KUKA KRL program: EPS_2_25694_GD03_A_20260114065902.src

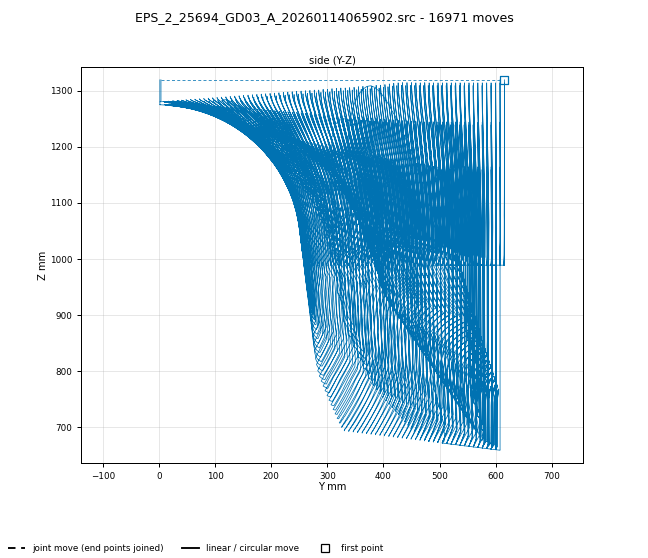
[picture p0: tool path of EPS_2_25694_GD03_A_20260114065902.src, 16971 of 16973 moves have a stored position in this frame; points joined in program order, loops and branches not executed]
&ACCESS RVP
&REL 4
&COMMENT QRS 19112012
&PARAM EDITMASK = *
DEF PART()
EXT BAS (BAS_COMMAND :IN,REAL :IN )
INT I
BAS (#INITMOV,0 )

;KUKA QRS Post kuka4.cps  Date:22-06-2017 !

File_ID=2970

QRS_PRE_INIT()

;Init var - Until changes are made in qrs_pre_init
Outlet_Square_prg=0
Inlet_1_Square_prg=0
Inlet_2_Square_prg=0
Inlet_3_Square_prg=0
Inlet_4_Square_prg=0
Inlet_5_Square_prg=0

Outlet_1={X 0.000, Y 425.000, Z 1043.000, B 0.000, E1 0.000 }
Inlet_1={X 0.000, Y 466.000, Z 1011.000, B 0.000, E1 180.000 }
Inlet_2={X 0.000, Y 490.880, Z 930.000, B 0.000, E1 271.000 }
Outlet_1_type=533
Inlet_1_type=457
Inlet_2_type=299
;QRS#1=Sidecore dimensions
;QRS#2=525-21" Concrete
;QRS#3=450-18" Concrete
;QRS#4=300-12" PVC SDR 35
;QRS#5=
;QRS#6=
;QRS#7=
;QRS#8=
;QRS#9=S306-32
;QRS#10=28A PSX-2
;QRS#11=16M PSX
;QRS#12=
;QRS#13=
;QRS#14=
;QRS#15=
;QRS#16=1220x127x1676 5,5'
;QRS#17=EPS Height
;QRS#18=1309,5
;QRS#19=*
;QRS#20= UPDATED VERSION 22-06-2017
;QRS#21=*
Outlet_Square=0250
Inlet_1_Square=0250
Inlet_2_Square=0150
Inlet_3_Square=0
Inlet_4_Square=0
Inlet_5_Square=0
Mill_Square=1
Outlet_Square_Prg=263
Inlet_1_Square_prg=274
Inlet_2_Square_prg=206

QRS_INIT()

$ADVANCE=5

; T1
PTP {E1 172.532,E2 172.532}
PTP {X 0,Y 615.614,A -85,B 0,C 180,E1 172.532,E2 172.532,E3 0,E4 0,E5 0,E6 0}
QRS_SPEED_INIT()
LIN {X 0,Y 615.614,Z 1319.5,A -85,B 0,C 180,E1 172.532,E2 172.532,E3 0,E4 0,E5 0,E6 0} C_VEL
LIN {X 0,Y 615.614,Z 991.03,A -85,B 0,C 180,E1 172.532,E2 172.532} C_VEL
LIN {X 0,Y 615.559,Z 989.03,A -85,B 0,C 180,E1 172.718,E2 172.718} C_VEL
LIN {X 0,Y 615.859,Z 989.03,A -85,B 0,C 180,E1 176.52,E2 176.52} C_VEL
LIN {X 0,Y 615.859,Z 989.03,A -85,B 0,C 180,E1 181.159,E2 181.159} C_VEL
LIN {X 0,Y 615.851,Z 989.03,A -85,B 0,C 180,E1 185.807,E2 185.807} C_VEL
LIN {X 0,Y 615.828,Z 989.03,A -85,B 0,C 180,E1 190.493,E2 190.493} C_VEL
LIN {X 0,Y 615.82,Z 989.03,A -85,B 0,C 180,E1 195.252,E2 195.252} C_VEL
LIN {X 0,Y 615.788,Z 989.03,A -85,B 0,C 180,E1 200.122,E2 200.122} C_VEL
LIN {X 0,Y 615.781,Z 989.03,A -85,B 0,C 180,E1 205.149,E2 205.149} C_VEL
LIN {X 0,Y 615.249,Z 989.03,A -85,B 0,C 180,E1 207.765,E2 207.765} C_VEL
LIN {X 0,Y 615.753,Z 989.03,A -85,B 0,C 180,E1 210.394,E2 210.394} C_VEL
LIN {X 0,Y 615.151,Z 989.03,A -85,B 0,C 180,E1 213.846,E2 213.846} C_VEL
LIN {X 0,Y 615.688,Z 989.03,A -85,B 0,C 180,E1 215.941,E2 215.941} C_VEL
LIN {X 0,Y 615.425,Z 989.03,A -85,B 0,C 180,E1 217.845,E2 217.845} C_VEL
LIN {X 0,Y 615.375,Z 989.03,A -85,B 0,C 180,E1 218.884,E2 218.884} C_VEL
LIN {X 0,Y 615.648,Z 989.03,A -85,B 0,C 180,E1 221.505,E2 221.505} C_VEL
LIN {X 0,Y 615.679,Z 989.03,A -85,B 0,C 180,E1 225.105,E2 225.105} C_VEL
LIN {X 0,Y 615.276,Z 989.03,A -85,B 0,C 180,E1 228.536,E2 228.536} C_VEL
LIN {X 0,Y 615.663,Z 989.03,A -85,B 0,C 180,E1 231.138,E2 231.138} C_VEL
LIN {X 0,Y 615.643,Z 989.03,A -85,B 0,C 180,E1 236.087,E2 236.087} C_VEL
LIN {X 0,Y 615.764,Z 989.03,A -85,B 0,C 180,E1 236.88,E2 236.88} C_VEL
LIN {X 0,Y 615.664,Z 989.03,A -85,B 0,C 180,E1 239.602,E2 239.602} C_VEL
LIN {X 0,Y 615.562,Z 989.03,A -85,B 0,C 180,E1 240.511,E2 240.511} C_VEL
LIN {X 0,Y 615.283,Z 989.03,A -85,B 0,C 180,E1 240.561,E2 240.561} C_VEL
LIN {X 0,Y 615.22,Z 991.782,A -85,B 0,C 180,E1 240.607,E2 240.607} C_VEL
LIN {X 0,Y 615.436,Z 1058.584,A -85,B 0,C 180,E1 241.501,E2 241.501} C_VEL
LIN {X 0,Y 615.528,Z 1069.337,A -85,B 0,C 180,E1 241.681,E2 241.681} C_VEL
LIN {X 0,Y 615.536,Z 1083.634,A -85,B 0,C 180,E1 241.987,E2 241.987} C_VEL
LIN {X 0,Y 615.498,Z 1092.536,A -85,B 0,C 180,E1 242.211,E2 242.211} C_VEL
LIN {X 0,Y 615.673,Z 1108.534,A -85,B 0,C 180,E1 242.706,E2 242.706} C_VEL
LIN {X 0,Y 615.633,Z 1120.967,A -85,B 0,C 180,E1 243.152,E2 243.152} C_VEL
LIN {X 0,Y 615.564,Z 1130.883,A -85,B 0,C 180,E1 243.554,E2 243.554} C_VEL
LIN {X 0,Y 615.7,Z 1146.603,A -85,B 0,C 180,E1 244.287,E2 244.287} C_VEL
LIN {X 0,Y 615.683,Z 1158.953,A -85,B 0,C 180,E1 244.936,E2 244.936} C_VEL
LIN {X 0,Y 615.67,Z 1170.644,A -85,B 0,C 180,E1 245.618,E2 245.618} C_VEL
LIN {X 0,Y 615.71,Z 1182.425,A -85,B 0,C 180,E1 246.381,E2 246.381} C_VEL
LIN {X 0,Y 615.719,Z 1193.095,A -85,B 0,C 180,E1 247.135,E2 247.135} C_VEL
LIN {X 0,Y 615.707,Z 1204.396,A -85,B 0,C 180,E1 248.012,E2 248.012} C_VEL
LIN {X 0,Y 615.705,Z 1213.657,A -85,B 0,C 180,E1 248.792,E2 248.792} C_VEL
LIN {X 0,Y 615.754,Z 1223.793,A -85,B 0,C 180,E1 249.723,E2 249.723} C_VEL
LIN {X 0,Y 615.723,Z 1233.057,A -85,B 0,C 180,E1 250.647,E2 250.647} C_VEL
LIN {X 0,Y 615.68,Z 1241.424,A -85,B 0,C 180,E1 251.549,E2 251.549} C_VEL
LIN {X 0,Y 615.758,Z 1249.778,A -85,B 0,C 180,E1 252.532,E2 252.532} C_VEL
LIN {X 0,Y 615.711,Z 1257.683,A -85,B 0,C 180,E1 253.542,E2 253.542} C_VEL
LIN {X 0,Y 615.578,Z 1264.428,A -85,B 0,C 180,E1 254.473,E2 254.473} C_VEL
LIN {X 0,Y 615.673,Z 1272.062,A -85,B 0,C 180,E1 255.645,E2 255.645} C_VEL
LIN {X 0,Y 615.813,Z 1277.439,A -85,B 0,C 180,E1 256.544,E2 256.544} C_VEL
LIN {X 0,Y 615.579,Z 1283.911,A -85,B 0,C 180,E1 257.728,E2 257.728} C_VEL
LIN {X 0,Y 615.618,Z 1289.625,A -85,B 0,C 180,E1 258.914,E2 258.914} C_VEL
LIN {X 0,Y 615.829,Z 1294.635,A -85,B 0,C 180,E1 260.097,E2 260.097} C_VEL
LIN {X 0,Y 615.605,Z 1299.064,A -85,B 0,C 180,E1 261.268,E2 261.268} C_VEL
LIN {X 0,Y 615.656,Z 1303.46,A -85,B 0,C 180,E1 262.657,E2 262.657} C_VEL
LIN {X 0,Y 615.79,Z 1306.368,A -85,B 0,C 180,E1 263.748,E2 263.748} C_VEL
LIN {X 0,Y 615.529,Z 1309.384,A -85,B 0,C 180,E1 265.123,E2 265.123} C_VEL
LIN {X 0,Y 615.632,Z 1311.594,A -85,B 0,C 180,E1 266.519,E2 266.519} C_VEL
LIN {X 0,Y 615.819,Z 1312.67,A -85,B 0,C 180,E1 267.449,E2 267.449} C_VEL
LIN {X 0,Y 615.544,Z 1313.716,A -85,B 0,C 180,E1 268.84,E2 268.84} C_VEL
LIN {X 0,Y 615.841,Z 1313.659,A -85,B 0,C 180,E1 271.16,E2 271.16} C_VEL
LIN {X 0,Y 615.625,Z 1313.07,A -85,B 0,C 180,E1 272.088,E2 272.088} C_VEL
LIN {X 0,Y 615.537,Z 1311.61,A -85,B 0,C 180,E1 273.482,E2 273.482} C_VEL
LIN {X 0,Y 615.808,Z 1309.332,A -85,B 0,C 180,E1 274.876,E2 274.876} C_VEL
LIN {X 0,Y 615.603,Z 1306.408,A -85,B 0,C 180,E1 276.25,E2 276.25} C_VEL
LIN {X 0,Y 615.617,Z 1303.276,A -85,B 0,C 180,E1 277.415,E2 277.415} C_VEL
LIN {X 0,Y 615.787,Z 1299.033,A -85,B 0,C 180,E1 278.73,E2 278.73} C_VEL
LIN {X 0,Y 615.576,Z 1294.668,A -85,B 0,C 180,E1 279.908,E2 279.908} C_VEL
LIN {X 0,Y 615.636,Z 1289.619,A -85,B 0,C 180,E1 281.087,E2 281.087} C_VEL
LIN {X 0,Y 615.81,Z 1283.879,A -85,B 0,C 180,E1 282.268,E2 282.268} C_VEL
LIN {X 0,Y 615.629,Z 1277.451,A -85,B 0,C 180,E1 283.461,E2 283.461} C_VEL
LIN {X 0,Y 615.698,Z 1270.19,A -85,B 0,C 180,E1 284.655,E2 284.655} C_VEL
LIN {X 0,Y 615.81,Z 1264.632,A -85,B 0,C 180,E1 285.488,E2 285.488} C_VEL
LIN {X 0,Y 615.663,Z 1255.195,A -85,B 0,C 180,E1 286.791,E2 286.791} C_VEL
LIN {X 0,Y 615.737,Z 1246.602,A -85,B 0,C 180,E1 287.853,E2 287.853} C_VEL
LIN {X 0,Y 615.77,Z 1238.406,A -85,B 0,C 180,E1 288.785,E2 288.785} C_VEL
LIN {X 0,Y 615.695,Z 1228.516,A -85,B 0,C 180,E1 289.817,E2 289.817} C_VEL
LIN {X 0,Y 615.712,Z 1220.53,A -85,B 0,C 180,E1 290.589,E2 290.589} C_VEL
LIN {X 0,Y 615.743,Z 1210.026,A -85,B 0,C 180,E1 291.519,E2 291.519} C_VEL
LIN {X 0,Y 615.702,Z 1200.055,A -85,B 0,C 180,E1 292.335,E2 292.335} C_VEL
LIN {X 0,Y 615.701,Z 1190.279,A -85,B 0,C 180,E1 293.072,E2 293.072} C_VEL
LIN {X 0,Y 615.684,Z 1178.611,A -85,B 0,C 180,E1 293.875,E2 293.875} C_VEL
LIN {X 0,Y 615.706,Z 1166.571,A -85,B 0,C 180,E1 294.624,E2 294.624} C_VEL
LIN {X 0,Y 615.665,Z 1155.875,A -85,B 0,C 180,E1 295.234,E2 295.234} C_VEL
LIN {X 0,Y 615.663,Z 1145.005,A -85,B 0,C 180,E1 295.796,E2 295.796} C_VEL
LIN {X 0,Y 615.699,Z 1130.858,A -85,B 0,C 180,E1 296.441,E2 296.441} C_VEL
LIN {X 0,Y 615.618,Z 1117.653,A -85,B 0,C 180,E1 296.972,E2 296.972} C_VEL
LIN {X 0,Y 615.557,Z 1108.505,A -85,B 0,C 180,E1 297.3,E2 297.3} C_VEL
LIN {X 0,Y 615.621,Z 1091.817,A -85,B 0,C 180,E1 297.801,E2 297.801} C_VEL
LIN {X 0,Y 615.426,Z 1077.854,A -85,B 0,C 180,E1 298.151,E2 298.151} C_VEL
LIN {X 0,Y 615.621,Z 1067.72,A -85,B 0,C 180,E1 298.346,E2 298.346} C_VEL
LIN {X 0,Y 615.638,Z 1052.258,A -85,B 0,C 180,E1 298.581,E2 298.581} C_VEL
LIN {X 0,Y 615.238,Z 989.03,A -85,B 0,C 180,E1 299.431,E2 299.431} C_VEL
LIN {X 0,Y 615.837,Z 989.03,A -85,B 0,C 180,E1 300.389,E2 300.389} C_VEL
LIN {X 0,Y 615.688,Z 989.03,A -85,B 0,C 180,E1 305.941,E2 305.941} C_VEL
LIN {X 0,Y 615.421,Z 989.03,A -85,B 0,C 180,E1 307.843,E2 307.843} C_VEL
LIN {X 0,Y 615.376,Z 989.03,A -85,B 0,C 180,E1 308.884,E2 308.884} C_VEL
LIN {X 0,Y 615.654,Z 989.03,A -85,B 0,C 180,E1 311.504,E2 311.504} C_VEL
LIN {X 0,Y 615.673,Z 989.03,A -85,B 0,C 180,E1 315.105,E2 315.105} C_VEL
LIN {X 0,Y 615.274,Z 989.03,A -85,B 0,C 180,E1 318.536,E2 318.536} C_VEL
LIN {X 0,Y 615.659,Z 989.03,A -85,B 0,C 180,E1 321.137,E2 321.137} C_VEL
LIN {X 0,Y 615.644,Z 989.03,A -85,B 0,C 180,E1 326.087,E2 326.087} C_VEL
LIN {X 0,Y 615.729,Z 989.03,A -85,B 0,C 180,E1 326.877,E2 326.877} C_VEL
LIN {X 0,Y 615.562,Z 989.03,A -85,B 0,C 180,E1 330.515,E2 330.515} C_VEL
LIN {X 0,Y 615.527,Z 989.03,A -85,B 0,C 180,E1 332.249,E2 332.249} C_VEL
LIN {X 0,Y 615.437,Z 989.03,A -85,B 0,C 180,E1 335.666,E2 335.666} C_VEL
LIN {X 0,Y 615.626,Z 989.03,A -85,B 0,C 180,E1 337.381,E2 337.381} C_VEL
LIN {X 0,Y 615.841,Z 989.03,A -85,B 0,C 180,E1 341.59,E2 341.59} C_VEL
LIN {X 0,Y 615.456,Z 989.03,A -85,B 0,C 180,E1 341.764,E2 341.764} C_VEL
LIN {X 0,Y 614.755,Z 989.116,A -85,B 0,C 180,E1 341.896,E2 341.896} C_VEL
LIN {X 0,Y 615.625,Z 991.909,A -85,B 0,C 180,E1 341.954,E2 341.954} C_VEL
LIN {X 0,Y 615.739,Z 1013.185,A -85,B 0,C 180,E1 342.225,E2 342.225} C_VEL
LIN {X 0,Y 615.775,Z 1024.708,A -85,B 0,C 180,E1 342.442,E2 342.442} C_VEL
LIN {X 0,Y 615.741,Z 1034.023,A -85,B 0,C 180,E1 342.673,E2 342.673} C_VEL
LIN {X 0,Y 615.81,Z 1042.538,A -85,B 0,C 180,E1 342.931,E2 342.931} C_VEL
LIN {X 0,Y 615.79,Z 1050.998,A -85,B 0,C 180,E1 343.231,E2 343.231} C_VEL
LIN {X 0,Y 615.791,Z 1058.355,A -85,B 0,C 180,E1 343.53,E2 343.53} C_VEL
LIN {X 0,Y 615.825,Z 1066.455,A -85,B 0,C 180,E1 343.905,E2 343.905} C_VEL
LIN {X 0,Y 615.822,Z 1075.021,A -85,B 0,C 180,E1 344.351,E2 344.351} C_VEL
LIN {X 0,Y 615.806,Z 1084.215,A -85,B 0,C 180,E1 344.898,E2 344.898} C_VEL
LIN {X 0,Y 615.816,Z 1091.974,A -85,B 0,C 180,E1 345.423,E2 345.423} C_VEL
LIN {X 0,Y 615.835,Z 1098.953,A -85,B 0,C 180,E1 345.947,E2 345.947} C_VEL
LIN {X 0,Y 615.816,Z 1106.145,A -85,B 0,C 180,E1 346.543,E2 346.543} C_VEL
LIN {X 0,Y 615.78,Z 1114.174,A -85,B 0,C 180,E1 347.287,E2 347.287} C_VEL
LIN {X 0,Y 615.817,Z 1121.188,A -85,B 0,C 180,E1 348.029,E2 348.029} C_VEL
LIN {X 0,Y 615.768,Z 1127.476,A -85,B 0,C 180,E1 348.768,E2 348.768} C_VEL
LIN {X 0,Y 615.713,Z 1134.153,A -85,B 0,C 180,E1 349.652,E2 349.652} C_VEL
LIN {X 0,Y 615.776,Z 1139,A -85,B 0,C 180,E1 350.389,E2 350.389} C_VEL
LIN {X 0,Y 615.832,Z 1142.522,A -85,B 0,C 180,E1 350.978,E2 350.978} C_VEL
LIN {X 0,Y 615.728,Z 1147.185,A -85,B 0,C 180,E1 351.856,E2 351.856} C_VEL
LIN {X 0,Y 615.739,Z 1150.609,A -85,B 0,C 180,E1 352.595,E2 352.595} C_VEL
LIN {X 0,Y 615.825,Z 1155.059,A -85,B 0,C 180,E1 353.73,E2 353.73} C_VEL
LIN {X 0,Y 615.692,Z 1157.976,A -85,B 0,C 180,E1 354.658,E2 354.658} C_VEL
LIN {X 0,Y 615.708,Z 1160.282,A -85,B 0,C 180,E1 355.589,E2 355.589} C_VEL
LIN {X 0,Y 615.833,Z 1162.004,A -85,B 0,C 180,E1 356.52,E2 356.52} C_VEL
LIN {X 0,Y 615.707,Z 1163.226,A -85,B 0,C 180,E1 357.448,E2 357.448} C_VEL
LIN {X 0,Y 615.681,Z 1163.573,A -85,B 0,C 180,E1 357.912,E2 357.912} C_VEL
LIN {X 0,Y 615.746,Z 1163.924,A -85,B 0,C 180,E1 358.84,E2 358.84} C_VEL
LIN {X 0,Y 615.836,Z 1163.85,A -85,B 0,C 180,E1 359.304,E2 359.304} C_VEL
LIN {X 0,Y 615.747,Z 1163.395,A -85,B 0,C 180,E1 360.232,E2 360.232} C_VEL
LIN {X 0,Y 615.728,Z 1162.397,A -85,B 0,C 180,E1 361.16,E2 361.16} C_VEL
LIN {X 0,Y 615.787,Z 1161.624,A -85,B 0,C 180,E1 361.623,E2 361.623} C_VEL
LIN {X 0,Y 615.773,Z 1159.77,A -85,B 0,C 180,E1 362.552,E2 362.552} C_VEL
LIN {X 0,Y 615.679,Z 1157.339,A -85,B 0,C 180,E1 363.481,E2 363.481} C_VEL
LIN {X 0,Y 615.756,Z 1154.217,A -85,B 0,C 180,E1 364.411,E2 364.411} C_VEL
LIN {X 0,Y 615.844,Z 1152.461,A -85,B 0,C 180,E1 364.875,E2 364.875} C_VEL
LIN {X 0,Y 615.752,Z 1148.382,A -85,B 0,C 180,E1 365.808,E2 365.808} C_VEL
LIN {X 0,Y 615.736,Z 1143.294,A -85,B 0,C 180,E1 366.795,E2 366.795} C_VEL
LIN {X 0,Y 615.848,Z 1138.485,A -85,B 0,C 180,E1 367.603,E2 367.603} C_VEL
LIN {X 0,Y 615.764,Z 1132.854,A -85,B 0,C 180,E1 368.437,E2 368.437} C_VEL
LIN {X 0,Y 615.762,Z 1127.247,A -85,B 0,C 180,E1 369.17,E2 369.17} C_VEL
LIN {X 0,Y 615.833,Z 1120.977,A -85,B 0,C 180,E1 369.904,E2 369.904} C_VEL
LIN {X 0,Y 615.792,Z 1113.996,A -85,B 0,C 180,E1 370.641,E2 370.641} C_VEL
LIN {X 0,Y 615.785,Z 1106.006,A -85,B 0,C 180,E1 371.379,E2 371.379} C_VEL
LIN {X 0,Y 615.819,Z 1098.86,A -85,B 0,C 180,E1 371.971,E2 371.971} C_VEL
LIN {X 0,Y 615.818,Z 1089.866,A -85,B 0,C 180,E1 372.638,E2 372.638} C_VEL
LIN {X 0,Y 615.81,Z 1080.602,A -85,B 0,C 180,E1 373.233,E2 373.233} C_VEL
LIN {X 0,Y 615.807,Z 1072.771,A -85,B 0,C 180,E1 373.68,E2 373.68} C_VEL
LIN {X 0,Y 615.825,Z 1065.468,A -85,B 0,C 180,E1 374.053,E2 374.053} C_VEL
LIN {X 0,Y 615.826,Z 1057.238,A -85,B 0,C 180,E1 374.427,E2 374.427} C_VEL
LIN {X 0,Y 615.789,Z 1046.747,A -85,B 0,C 180,E1 374.84,E2 374.84} C_VEL
LIN {X 0,Y 615.798,Z 1036.447,A -85,B 0,C 180,E1 375.168,E2 375.168} C_VEL
LIN {X 0,Y 615.816,Z 1027.25,A -85,B 0,C 180,E1 375.408,E2 375.408} C_VEL
LIN {X 0,Y 615.796,Z 1017.993,A -85,B 0,C 180,E1 375.602,E2 375.602} C_VEL
LIN {X 0,Y 615.588,Z 1007.058,A -85,B 0,C 180,E1 375.776,E2 375.776} C_VEL
LIN {X 0,Y 614.781,Z 993.128,A -85,B 0,C 180,E1 375.965,E2 375.965} C_VEL
LIN {X 0,Y 614.429,Z 989.03,A -85,B 0,C 180,E1 376.026,E2 376.026} C_VEL
LIN {X 0,Y 615.422,Z 989.03,A -85,B 0,C 180,E1 376.144,E2 376.144} C_VEL
LIN {X 0,Y 615.843,Z 989.03,A -85,B 0,C 180,E1 376.464,E2 376.464} C_VEL
LIN {X 0,Y 615.798,Z 989.03,A -85,B 0,C 180,E1 377.993,E2 377.993} C_VEL
LIN {X 0,Y 615.789,Z 989.03,A -85,B 0,C 180,E1 382.612,E2 382.612} C_VEL
LIN {X 0,Y 615.245,Z 989.03,A -85,B 0,C 180,E1 385.172,E2 385.172} C_VEL
LIN {X 0,Y 615.749,Z 989.03,A -85,B 0,C 180,E1 387.741,E2 387.741} C_VEL
LIN {X 0,Y 615.174,Z 989.03,A -85,B 0,C 180,E1 390.425,E2 390.425} C_VEL
LIN {X 0,Y 615.699,Z 989.03,A -85,B 0,C 180,E1 393.125,E2 393.125} C_VEL
LIN {X 0,Y 615.641,Z 989.03,A -85,B 0,C 180,E1 393.913,E2 393.913} C_VEL
LIN {X 0,Y 615.654,Z 989.03,A -85,B 0,C 180,E1 398.864,E2 398.864} C_VEL
LIN {X 0,Y 615.253,Z 989.03,A -85,B 0,C 180,E1 401.942,E2 401.942} C_VEL
LIN {X 0,Y 615.678,Z 989.03,A -85,B 0,C 180,E1 404.895,E2 404.895} C_VEL
LIN {X 0,Y 615.657,Z 989.03,A -85,B 0,C 180,E1 408.496,E2 408.496} C_VEL
LIN {X 0,Y 615.375,Z 989.03,A -85,B 0,C 180,E1 411.116,E2 411.116} C_VEL
LIN {X 0,Y 615.427,Z 989.03,A -85,B 0,C 180,E1 412.156,E2 412.156} C_VEL
LIN {X 0,Y 615.691,Z 989.03,A -85,B 0,C 180,E1 414.059,E2 414.059} C_VEL
LIN {X 0,Y 615.146,Z 989.03,A -85,B 0,C 180,E1 416.842,E2 416.842} C_VEL
LIN {X 0,Y 615.732,Z 989.03,A -85,B 0,C 180,E1 419.605,E2 419.605} C_VEL
LIN {X 0,Y 615.223,Z 989.03,A -85,B 0,C 180,E1 422.234,E2 422.234} C_VEL
LIN {X 0,Y 615.271,Z 989.03,A -85,B 0,C 180,E1 424.829,E2 424.829} C_VEL
LIN {X 0,Y 614.55,Z 989.03,A -85,B 0,C 180,E1 424.916,E2 424.916} C_VEL
LIN {X 0,Y 615.319,Z 993.108,A -85,B 0,C 180,E1 425.004,E2 425.004} C_VEL
LIN {X 0,Y 615.55,Z 999.968,A -85,B 0,C 180,E1 425.1,E2 425.1} C_VEL
LIN {X 0,Y 615.616,Z 1023.023,A -85,B 0,C 180,E1 425.405,E2 425.405} C_VEL
LIN {X 0,Y 615.531,Z 1033.042,A -85,B 0,C 180,E1 425.57,E2 425.57} C_VEL
LIN {X 0,Y 615.676,Z 1043.873,A -85,B 0,C 180,E1 425.805,E2 425.805} C_VEL
LIN {X 0,Y 615.68,Z 1055.337,A -85,B 0,C 180,E1 426.101,E2 426.101} C_VEL
LIN {X 0,Y 615.609,Z 1065.34,A -85,B 0,C 180,E1 426.402,E2 426.402} C_VEL
LIN {X 0,Y 615.758,Z 1076.758,A -85,B 0,C 180,E1 426.812,E2 426.812} C_VEL
LIN {X 0,Y 615.773,Z 1088.067,A -85,B 0,C 180,E1 427.272,E2 427.272} C_VEL
LIN {X 0,Y 615.72,Z 1098.214,A -85,B 0,C 180,E1 427.735,E2 427.735} C_VEL
LIN {X 0,Y 615.726,Z 1109.631,A -85,B 0,C 180,E1 428.324,E2 428.324} C_VEL
LIN {X 0,Y 615.756,Z 1120.432,A -85,B 0,C 180,E1 428.948,E2 428.948} C_VEL
LIN {X 0,Y 615.751,Z 1130.175,A -85,B 0,C 180,E1 429.568,E2 429.568} C_VEL
LIN {X 0,Y 615.753,Z 1139.056,A -85,B 0,C 180,E1 430.185,E2 430.185} C_VEL
LIN {X 0,Y 615.747,Z 1149.104,A -85,B 0,C 180,E1 430.953,E2 430.953} C_VEL
LIN {X 0,Y 615.776,Z 1157.253,A -85,B 0,C 180,E1 431.632,E2 431.632} C_VEL
LIN {X 0,Y 615.74,Z 1166.041,A -85,B 0,C 180,E1 432.428,E2 432.428} C_VEL
LIN {X 0,Y 615.696,Z 1173.201,A -85,B 0,C 180,E1 433.13,E2 433.13} C_VEL
LIN {X 0,Y 615.74,Z 1181.142,A -85,B 0,C 180,E1 433.981,E2 433.981} C_VEL
LIN {X 0,Y 615.808,Z 1187.743,A -85,B 0,C 180,E1 434.748,E2 434.748} C_VEL
LIN {X 0,Y 615.677,Z 1194.859,A -85,B 0,C 180,E1 435.644,E2 435.644} C_VEL
LIN {X 0,Y 615.669,Z 1201.329,A -85,B 0,C 180,E1 436.54,E2 436.54} C_VEL
LIN {X 0,Y 615.797,Z 1207.201,A -85,B 0,C 180,E1 437.435,E2 437.435} C_VEL
LIN {X 0,Y 615.687,Z 1212.564,A -85,B 0,C 180,E1 438.322,E2 438.322} C_VEL
LIN {X 0,Y 615.612,Z 1218.867,A -85,B 0,C 180,E1 439.503,E2 439.503} C_VEL
LIN {X 0,Y 615.726,Z 1223.092,A -85,B 0,C 180,E1 440.388,E2 440.388} C_VEL
LIN {X 0,Y 615.757,Z 1226.863,A -85,B 0,C 180,E1 441.27,E2 441.27} C_VEL
LIN {X 0,Y 615.619,Z 1231.735,A -85,B 0,C 180,E1 442.581,E2 442.581} C_VEL
LIN {X 0,Y 615.76,Z 1235.305,A -85,B 0,C 180,E1 443.75,E2 443.75} C_VEL
LIN {X 0,Y 615.83,Z 1236.478,A -85,B 0,C 180,E1 444.193,E2 444.193} C_VEL
LIN {X 0,Y 615.634,Z 1238.723,A -85,B 0,C 180,E1 445.123,E2 445.123} C_VEL
LIN {X 0,Y 615.613,Z 1241.326,A -85,B 0,C 180,E1 446.518,E2 446.518} C_VEL
LIN {X 0,Y 615.786,Z 1242.496,A -85,B 0,C 180,E1 447.448,E2 447.448} C_VEL
LIN {X 0,Y 615.781,Z 1243.003,A -85,B 0,C 180,E1 447.912,E2 447.912} C_VEL
LIN {X 0,Y 615.602,Z 1243.694,A -85,B 0,C 180,E1 448.84,E2 448.84} C_VEL
LIN {X 0,Y 615.58,Z 1243.938,A -85,B 0,C 180,E1 449.768,E2 449.768} C_VEL
LIN {X 0,Y 615.835,Z 1243.585,A -85,B 0,C 180,E1 451.159,E2 451.159} C_VEL
LIN {X 0,Y 615.642,Z 1242.418,A -85,B 0,C 180,E1 452.552,E2 452.552} C_VEL
LIN {X 0,Y 615.679,Z 1241.163,A -85,B 0,C 180,E1 453.481,E2 453.481} C_VEL
LIN {X 0,Y 615.845,Z 1239.506,A -85,B 0,C 180,E1 454.409,E2 454.409} C_VEL
LIN {X 0,Y 615.652,Z 1237.512,A -85,B 0,C 180,E1 455.342,E2 455.342} C_VEL
LIN {X 0,Y 615.594,Z 1233.883,A -85,B 0,C 180,E1 456.66,E2 456.66} C_VEL
LIN {X 0,Y 615.746,Z 1231.125,A -85,B 0,C 180,E1 457.509,E2 457.509} C_VEL
LIN {X 0,Y 615.732,Z 1227.668,A -85,B 0,C 180,E1 458.437,E2 458.437} C_VEL
LIN {X 0,Y 615.616,Z 1222.717,A -85,B 0,C 180,E1 459.613,E2 459.613} C_VEL
LIN {X 0,Y 615.757,Z 1216.89,A -85,B 0,C 180,E1 460.789,E2 460.789} C_VEL
LIN {X 0,Y 615.751,Z 1212.041,A -85,B 0,C 180,E1 461.675,E2 461.675} C_VEL
LIN {X 0,Y 615.662,Z 1206.676,A -85,B 0,C 180,E1 462.567,E2 462.567} C_VEL
LIN {X 0,Y 615.744,Z 1199.684,A -85,B 0,C 180,E1 463.607,E2 463.607} C_VEL
LIN {X 0,Y 615.79,Z 1193.056,A -85,B 0,C 180,E1 464.502,E2 464.502} C_VEL
LIN {X 0,Y 615.686,Z 1184.706,A -85,B 0,C 180,E1 465.525,E2 465.525} C_VEL
LIN {X 0,Y 615.719,Z 1177.714,A -85,B 0,C 180,E1 466.307,E2 466.307} C_VEL
LIN {X 0,Y 615.786,Z 1169.333,A -85,B 0,C 180,E1 467.163,E2 467.163} C_VEL
LIN {X 0,Y 615.745,Z 1161.914,A -85,B 0,C 180,E1 467.866,E2 467.866} C_VEL
LIN {X 0,Y 615.74,Z 1153.893,A -85,B 0,C 180,E1 468.567,E2 468.567} C_VEL
LIN {X 0,Y 615.749,Z 1144.041,A -85,B 0,C 180,E1 469.353,E2 469.353} C_VEL
LIN {X 0,Y 615.758,Z 1134.53,A -85,B 0,C 180,E1 470.045,E2 470.045} C_VEL
LIN {X 0,Y 615.741,Z 1125.249,A -85,B 0,C 180,E1 470.664,E2 470.664} C_VEL
LIN {X 0,Y 615.704,Z 1114.982,A -85,B 0,C 180,E1 471.286,E2 471.286} C_VEL
LIN {X 0,Y 615.745,Z 1105.029,A -85,B 0,C 180,E1 471.83,E2 471.83} C_VEL
LIN {X 0,Y 615.75,Z 1094.442,A -85,B 0,C 180,E1 472.352,E2 472.352} C_VEL
LIN {X 0,Y 615.711,Z 1084.225,A -85,B 0,C 180,E1 472.804,E2 472.804} C_VEL
LIN {X 0,Y 615.644,Z 1074.601,A -85,B 0,C 180,E1 473.186,E2 473.186} C_VEL
LIN {X 0,Y 615.742,Z 1060.928,A -85,B 0,C 180,E1 473.641,E2 473.641} C_VEL
LIN {X 0,Y 615.686,Z 1049.242,A -85,B 0,C 180,E1 473.973,E2 473.973} C_VEL
LIN {X 0,Y 615.598,Z 1039.6,A -85,B 0,C 180,E1 474.208,E2 474.208} C_VEL
LIN {X 0,Y 615.732,Z 1027.492,A -85,B 0,C 180,E1 474.433,E2 474.433} C_VEL
LIN {X 0,Y 615.695,Z 1011.549,A -85,B 0,C 180,E1 474.658,E2 474.658} C_VEL
LIN {X 0,Y 615.559,Z 989.03,A -85,B 0,C 180,E1 474.957,E2 474.957} C_VEL
LIN {X 0,Y 615.871,Z 989.03,A -85,B 0,C 180,E1 475.144,E2 475.144} C_VEL
LIN {X 0,Y 615.789,Z 989.03,A -85,B 0,C 180,E1 477.738,E2 477.738} C_VEL
LIN {X 0,Y 615.172,Z 989.03,A -85,B 0,C 180,E1 480.425,E2 480.425} C_VEL
LIN {X 0,Y 615.698,Z 989.03,A -85,B 0,C 180,E1 483.124,E2 483.124} C_VEL
LIN {X 0,Y 615.634,Z 989.03,A -85,B 0,C 180,E1 483.911,E2 483.911} C_VEL
LIN {X 0,Y 615.655,Z 989.03,A -85,B 0,C 180,E1 488.862,E2 488.862} C_VEL
LIN {X 0,Y 615.25,Z 989.03,A -85,B 0,C 180,E1 491.941,E2 491.941} C_VEL
LIN {X 0,Y 615.662,Z 989.03,A -85,B 0,C 180,E1 494.893,E2 494.893} C_VEL
LIN {X 0,Y 615.652,Z 989.03,A -85,B 0,C 180,E1 498.495,E2 498.495} C_VEL
LIN {X 0,Y 615.376,Z 989.03,A -85,B 0,C 180,E1 501.116,E2 501.116} C_VEL
LIN {X 0,Y 615.421,Z 989.03,A -85,B 0,C 180,E1 502.155,E2 502.155} C_VEL
LIN {X 0,Y 615.691,Z 989.03,A -85,B 0,C 180,E1 504.059,E2 504.059} C_VEL
LIN {X 0,Y 615.155,Z 989.03,A -85,B 0,C 180,E1 506.842,E2 506.842} C_VEL
LIN {X 0,Y 615.752,Z 989.03,A -85,B 0,C 180,E1 509.606,E2 509.606} C_VEL
LIN {X 0,Y 615.246,Z 989.03,A -85,B 0,C 180,E1 512.235,E2 512.235} C_VEL
LIN {X 0,Y 615.777,Z 989.03,A -85,B 0,C 180,E1 514.851,E2 514.851} C_VEL
LIN {X 0,Y 615.802,Z 989.03,A -85,B 0,C 180,E1 519.878,E2 519.878} C_VEL
LIN {X 0,Y 615.521,Z 989.03,A -85,B 0,C 180,E1 522.321,E2 522.321} C_VEL
LIN {X 0,Y 615.633,Z 989.03,A -85,B 0,C 180,E1 524.744,E2 524.744} C_VEL
LIN {X 0,Y 615.813,Z 989.03,A -85,B 0,C 180,E1 527.139,E2 527.139} C_VEL
LIN {X 0,Y 615.852,Z 989.03,A -85,B 0,C 180,E1 531.857,E2 531.857} C_VEL
LIN {X 0,Y 615.559,Z 989.03,A -85,B 0,C 180,E1 532.718,E2 532.718} C_VEL
LIN {X 0,Y 611.546,Z 989.03,A -85,B 0,C 180,E1 534.305,E2 534.305} C_VEL
LIN {X 0,Y 607.682,Z 989.03,A -85,B 0,C 180,E1 535.913,E2 535.913} C_VEL
LIN {X 0,Y 607.871,Z 989.03,A -85,B 0,C 180,E1 541.423,E2 541.423} C_VEL
LIN {X 0,Y 607.672,Z 989.03,A -85,B 0,C 180,E1 546.643,E2 546.643} C_VEL
LIN {X 0,Y 607.611,Z 989.03,A -85,B 0,C 180,E1 551.46,E2 551.46} C_VEL
LIN {X 0,Y 607.672,Z 989.03,A -85,B 0,C 180,E1 555.852,E2 555.852} C_VEL
LIN {X 0,Y 607.795,Z 989.03,A -85,B 0,C 180,E1 560.339,E2 560.339} C_VEL
LIN {X 0,Y 607.801,Z 989.03,A -85,B 0,C 180,E1 564.964,E2 564.964} C_VEL
LIN {X 0,Y 607.622,Z 989.03,A -85,B 0,C 180,E1 569.78,E2 569.78} C_VEL
LIN {X 0,Y 607.654,Z 989.03,A -85,B 0,C 180,E1 576.582,E2 576.582} C_VEL
LIN {X 0,Y 607.603,Z 989.03,A -85,B 0,C 180,E1 582.108,E2 582.108} C_VEL
LIN {X 0,Y 607.282,Z 989.03,A -85,B 0,C 180,E1 587.865,E2 587.865} C_VEL
LIN {X 0,Y 607.29,Z 989.03,A -85,B 0,C 180,E1 592.666,E2 592.666} C_VEL
LIN {X 0,Y 607.715,Z 989.03,A -85,B 0,C 180,E1 597.588,E2 597.588} C_VEL
LIN {X 0,Y 607.683,Z 989.071,A -85,B 0,C 180,E1 600.17,E2 600.17} C_VEL
LIN {X 0,Y 608.593,Z 1077.308,A -85,B 0,C 180,E1 601.493,E2 601.493} C_VEL
LIN {X 0,Y 608.546,Z 1114.831,A -85,B 0,C 180,E1 602.587,E2 602.587} C_VEL
LIN {X 0,Y 608.426,Z 1150.852,A -85,B 0,C 180,E1 604.18,E2 604.18} C_VEL
LIN {X 0,Y 608.269,Z 1185.975,A -85,B 0,C 180,E1 606.325,E2 606.325} C_VEL
LIN {X 0,Y 608.11,Z 1218.031,A -85,B 0,C 180,E1 608.914,E2 608.914} C_VEL
LIN {X 0,Y 607.969,Z 1246.746,A -85,B 0,C 180,E1 611.928,E2 611.928} C_VEL
LIN {X 0,Y 607.832,Z 1271.206,A -85,B 0,C 180,E1 615.297,E2 615.297} C_VEL
LIN {X 0,Y 607.763,Z 1290.451,A -85,B 0,C 180,E1 618.908,E2 618.908} C_VEL
LIN {X 0,Y 607.782,Z 1303.724,A -85,B 0,C 180,E1 622.513,E2 622.513} C_VEL
LIN {X 0,Y 607.66,Z 1310.961,A -85,B 0,C 180,E1 625.73,E2 625.73} C_VEL
LIN {X 0,Y 607.698,Z 1314.088,A -85,B 0,C 180,E1 628.58,E2 628.58} C_VEL
LIN {X 0,Y 607.886,Z 1314.084,A -85,B 0,C 180,E1 631.425,E2 631.425} C_VEL
LIN {X 0,Y 607.906,Z 1309.751,A -85,B 0,C 180,E1 634.987,E2 634.987} C_VEL
LIN {X 0,Y 607.881,Z 1299.062,A -85,B 0,C 180,E1 638.929,E2 638.929} C_VEL
LIN {X 0,Y 607.909,Z 1283.434,A -85,B 0,C 180,E1 642.548,E2 642.548} C_VEL
LIN {X 0,Y 607.957,Z 1262.325,A -85,B 0,C 180,E1 646.033,E2 646.033} C_VEL
LIN {X 0,Y 608.032,Z 1236.031,A -85,B 0,C 180,E1 649.288,E2 649.288} C_VEL
LIN {X 0,Y 608.17,Z 1205.984,A -85,B 0,C 180,E1 652.142,E2 652.142} C_VEL
LIN {X 0,Y 608.325,Z 1172.835,A -85,B 0,C 180,E1 654.555,E2 654.555} C_VEL
LIN {X 0,Y 608.504,Z 1136.663,A -85,B 0,C 180,E1 656.515,E2 656.515} C_VEL
LIN {X 0,Y 608.576,Z 1099.62,A -85,B 0,C 180,E1 657.922,E2 657.922} C_VEL
LIN {X 0,Y 608.688,Z 1063.894,A -85,B 0,C 180,E1 658.762,E2 658.762} C_VEL
LIN {X 0,Y 607.95,Z 991.523,A -85,B 0,C 180,E1 659.783,E2 659.783} C_VEL
LIN {X 0,Y 607.642,Z 989.03,A -85,B 0,C 180,E1 659.951,E2 659.951} C_VEL
LIN {X 0,Y 607.624,Z 989.03,A -85,B 0,C 180,E1 666.591,E2 666.591} C_VEL
LIN {X 0,Y 607.611,Z 989.03,A -85,B 0,C 180,E1 672.115,E2 672.115} C_VEL
LIN {X 0,Y 607.279,Z 989.03,A -85,B 0,C 180,E1 677.864,E2 677.864} C_VEL
LIN {X 0,Y 607.288,Z 989.03,A -85,B 0,C 180,E1 682.676,E2 682.676} C_VEL
LIN {X 0,Y 607.592,Z 989.03,A -85,B 0,C 180,E1 687.618,E2 687.618} C_VEL
LIN {X 0,Y 607.606,Z 989.03,A -85,B 0,C 180,E1 691.845,E2 691.845} C_VEL
LIN {X 0,Y 607.53,Z 989.03,A -85,B 0,C 180,E1 698.126,E2 698.126} C_VEL
LIN {X 0,Y 607.263,Z 989.03,A -85,B 0,C 180,E1 701.67,E2 701.67} C_VEL
LIN {X 0,Y 608.203,Z 1029.893,A -85,B 0,C 180,E1 702.353,E2 702.353} C_VEL
LIN {X 0,Y 608.159,Z 1060.406,A -85,B 0,C 180,E1 703.421,E2 703.421} C_VEL
LIN {X 0,Y 608.085,Z 1088.207,A -85,B 0,C 180,E1 704.983,E2 704.983} C_VEL
LIN {X 0,Y 608.002,Z 1113.844,A -85,B 0,C 180,E1 707.093,E2 707.093} C_VEL
LIN {X 0,Y 607.884,Z 1133.81,A -85,B 0,C 180,E1 709.451,E2 709.451} C_VEL
LIN {X 0,Y 607.875,Z 1149.417,A -85,B 0,C 180,E1 712.153,E2 712.153} C_VEL
LIN {X 0,Y 607.821,Z 1159.547,A -85,B 0,C 180,E1 715.015,E2 715.015} C_VEL
LIN {X 0,Y 607.877,Z 1163.443,A -85,B 0,C 180,E1 717.154,E2 717.154} C_VEL
LIN {X 0,Y 607.884,Z 1164.12,A -85,B 0,C 180,E1 720,E2 720} C_VEL
LIN {X 0,Y 607.873,Z 1159.678,A -85,B 0,C 180,E1 722.845,E2 722.845} C_VEL
LIN {X 0,Y 607.92,Z 1149.698,A -85,B 0,C 180,E1 725.698,E2 725.698} C_VEL
LIN {X 0,Y 607.928,Z 1134.326,A -85,B 0,C 180,E1 728.385,E2 728.385} C_VEL
LIN {X 0,Y 607.992,Z 1114.722,A -85,B 0,C 180,E1 730.727,E2 730.727} C_VEL
LIN {X 0,Y 608.099,Z 1089.904,A -85,B 0,C 180,E1 732.813,E2 732.813} C_VEL
LIN {X 0,Y 608.192,Z 1061.092,A -85,B 0,C 180,E1 734.458,E2 734.458} C_VEL
LIN {X 0,Y 608.255,Z 1031.349,A -85,B 0,C 180,E1 735.519,E2 735.519} C_VEL
LIN {X 0,Y 607.379,Z 996.024,A -85,B 0,C 180,E1 736.144,E2 736.144} C_VEL
LIN {X 0,Y 606.905,Z 989.03,A -85,B 0,C 180,E1 736.252,E2 736.252} C_VEL
LIN {X 0,Y 607.883,Z 989.03,A -85,B 0,C 180,E1 737.33,E2 737.33} C_VEL
LIN {X 0,Y 607.608,Z 989.03,A -85,B 0,C 180,E1 743.412,E2 743.412} C_VEL
LIN {X 0,Y 607.682,Z 989.03,A -85,B 0,C 180,E1 748.15,E2 748.15} C_VEL
LIN {X 0,Y 607.803,Z 989.03,A -85,B 0,C 180,E1 753.105,E2 753.105} C_VEL
LIN {X 0,Y 607.485,Z 989.03,A -85,B 0,C 180,E1 759.635,E2 759.635} C_VEL
LIN {X 0,Y 607.533,Z 989.03,A -85,B 0,C 180,E1 765.93,E2 765.93} C_VEL
LIN {X 0,Y 607.425,Z 989.03,A -85,B 0,C 180,E1 770.361,E2 770.361} C_VEL
LIN {X 0,Y 607.427,Z 989.03,A -85,B 0,C 180,E1 775.149,E2 775.149} C_VEL
LIN {X 0,Y 607.562,Z 989.03,A -85,B 0,C 180,E1 780.372,E2 780.372} C_VEL
LIN {X 0,Y 607.342,Z 989.03,A -85,B 0,C 180,E1 784.594,E2 784.594} C_VEL
LIN {X 0,Y 608.425,Z 1027.708,A -85,B 0,C 180,E1 785.166,E2 785.166} C_VEL
LIN {X 0,Y 608.312,Z 1066.198,A -85,B 0,C 180,E1 786.132,E2 786.132} C_VEL
LIN {X 0,Y 608.306,Z 1102.564,A -85,B 0,C 180,E1 787.672,E2 787.672} C_VEL
LIN {X 0,Y 608.183,Z 1135.495,A -85,B 0,C 180,E1 789.67,E2 789.67} C_VEL
LIN {X 0,Y 608.064,Z 1165.144,A -85,B 0,C 180,E1 792.112,E2 792.112} C_VEL
LIN {X 0,Y 607.97,Z 1191.05,A -85,B 0,C 180,E1 794.959,E2 794.959} C_VEL
LIN {X 0,Y 607.872,Z 1212.781,A -85,B 0,C 180,E1 798.179,E2 798.179} C_VEL
LIN {X 0,Y 607.882,Z 1228.26,A -85,B 0,C 180,E1 801.431,E2 801.431} C_VEL
LIN {X 0,Y 607.79,Z 1239.079,A -85,B 0,C 180,E1 805.012,E2 805.012} C_VEL
LIN {X 0,Y 607.773,Z 1244.04,A -85,B 0,C 180,E1 808.574,E2 808.574} C_VEL
LIN {X 0,Y 607.901,Z 1243.98,A -85,B 0,C 180,E1 811.42,E2 811.42} C_VEL
LIN {X 0,Y 607.845,Z 1238.896,A -85,B 0,C 180,E1 814.982,E2 814.982} C_VEL
LIN {X 0,Y 607.865,Z 1227.947,A -85,B 0,C 180,E1 818.563,E2 818.563} C_VEL
LIN {X 0,Y 607.891,Z 1211.2,A -85,B 0,C 180,E1 821.997,E2 821.997} C_VEL
LIN {X 0,Y 607.942,Z 1189.666,A -85,B 0,C 180,E1 825.126,E2 825.126} C_VEL
LIN {X 0,Y 608.074,Z 1163.29,A -85,B 0,C 180,E1 827.976,E2 827.976} C_VEL
LIN {X 0,Y 608.19,Z 1132.907,A -85,B 0,C 180,E1 830.418,E2 830.418} C_VEL
LIN {X 0,Y 608.342,Z 1099.047,A -85,B 0,C 180,E1 832.417,E2 832.417} C_VEL
LIN {X 0,Y 608.481,Z 1062.358,A -85,B 0,C 180,E1 833.899,E2 833.899} C_VEL
LIN {X 0,Y 608.543,Z 1027.505,A -85,B 0,C 180,E1 834.742,E2 834.742} C_VEL
LIN {X 0,Y 607.93,Z 989.03,A -85,B 0,C 180,E1 835.297,E2 835.297} C_VEL
LIN {X 0,Y 607.318,Z 989.03,A -85,B 0,C 180,E1 839.796,E2 839.796} C_VEL
LIN {X 0,Y 607.798,Z 989.03,A -85,B 0,C 180,E1 843.105,E2 843.105} C_VEL
LIN {X 0,Y 607.504,Z 989.03,A -85,B 0,C 180,E1 849.648,E2 849.648} C_VEL
LIN {X 0,Y 607.514,Z 989.03,A -85,B 0,C 180,E1 855.936,E2 855.936} C_VEL
LIN {X 0,Y 607.425,Z 989.03,A -85,B 0,C 180,E1 860.363,E2 860.363} C_VEL
LIN {X 0,Y 607.423,Z 989.03,A -85,B 0,C 180,E1 865.155,E2 865.155} C_VEL
LIN {X 0,Y 607.568,Z 989.03,A -85,B 0,C 180,E1 870.374,E2 870.374} C_VEL
LIN {X 0,Y 607.798,Z 989.03,A -85,B 0,C 180,E1 875.036,E2 875.036} C_VEL
LIN {X 0,Y 607.646,Z 989.03,A -85,B 0,C 180,E1 881.167,E2 881.167} C_VEL
LIN {X 0,Y 607.915,Z 989.03,A -85,B 0,C 180,E1 887.092,E2 887.092} C_VEL
LIN {X 0,Y 607.622,Z 989.03,A -85,B 0,C 180,E1 892.868,E2 892.868} C_VEL
LIN {X 0,Y 607.682,Z 989.03,A -85,B 0,C 180,E1 895.913,E2 895.913} C_VEL
LIN {X 0,Y 606.354,Z 989.03,A -85,B 0,C 180,E1 896.726,E2 896.726} C_VEL
LIN {X 0,Y 599.656,Z 989.03,A -85,B 0,C 180,E1 898.937,E2 898.937} C_VEL
LIN {X 0,Y 599.577,Z 989.03,A -85,B 0,C 180,E1 899.146,E2 899.146} C_VEL
LIN {X 0,Y 599.627,Z 989.03,A -85,B 0,C 180,E1 902.885,E2 902.885} C_VEL
LIN {X 0,Y 599.611,Z 989.03,A -85,B 0,C 180,E1 907.229,E2 907.229} C_VEL
LIN {X 0,Y 599.668,Z 989.03,A -85,B 0,C 180,E1 911.613,E2 911.613} C_VEL
LIN {X 0,Y 599.702,Z 989.03,A -85,B 0,C 180,E1 916.068,E2 916.068} C_VEL
LIN {X 0,Y 599.565,Z 989.03,A -85,B 0,C 180,E1 921.376,E2 921.376} C_VEL
LIN {X 0,Y 599.793,Z 989.03,A -85,B 0,C 180,E1 925.321,E2 925.321} C_VEL
LIN {X 0,Y 599.54,Z 989.03,A -85,B 0,C 180,E1 931.159,E2 931.159} C_VEL
LIN {X 0,Y 599.665,Z 989.03,A -85,B 0,C 180,E1 937.151,E2 937.151} C_VEL
LIN {X 0,Y 599.573,Z 989.03,A -85,B 0,C 180,E1 943.126,E2 943.126} C_VEL
LIN {X 0,Y 599.423,Z 989.03,A -85,B 0,C 180,E1 949.118,E2 949.118} C_VEL
LIN {X 0,Y 599.303,Z 989.03,A -85,B 0,C 180,E1 953.679,E2 953.679} C_VEL
LIN {X 0,Y 599.771,Z 989.03,A -85,B 0,C 180,E1 958.108,E2 958.108} C_VEL
LIN {X 0,Y 599.902,Z 989.721,A -85,B 0,C 180,E1 959.752,E2 959.752} C_VEL
LIN {X 0,Y 601.477,Z 996.96,A -85,B 0,C 180,E1 959.937,E2 959.937} C_VEL
LIN {X 0,Y 601.62,Z 1077.369,A -85,B 0,C 180,E1 961.132,E2 961.132} C_VEL
LIN {X 0,Y 601.462,Z 1115.106,A -85,B 0,C 180,E1 962.246,E2 962.246} C_VEL
LIN {X 0,Y 601.182,Z 1150.872,A -85,B 0,C 180,E1 963.846,E2 963.846} C_VEL
LIN {X 0,Y 600.85,Z 1185.978,A -85,B 0,C 180,E1 966.014,E2 966.014} C_VEL
LIN {X 0,Y 600.538,Z 1217.063,A -85,B 0,C 180,E1 968.545,E2 968.545} C_VEL
LIN {X 0,Y 600.234,Z 1245.145,A -85,B 0,C 180,E1 971.497,E2 971.497} C_VEL
LIN {X 0,Y 599.991,Z 1269.766,A -85,B 0,C 180,E1 974.877,E2 974.877} C_VEL
LIN {X 0,Y 599.859,Z 1287.037,A -85,B 0,C 180,E1 978.024,E2 978.024} C_VEL
LIN {X 0,Y 599.845,Z 1300.31,A -85,B 0,C 180,E1 981.321,E2 981.321} C_VEL
LIN {X 0,Y 599.776,Z 1309.761,A -85,B 0,C 180,E1 984.951,E2 984.951} C_VEL
LIN {X 0,Y 599.799,Z 1314.09,A -85,B 0,C 180,E1 988.561,E2 988.561} C_VEL
LIN {X 0,Y 599.979,Z 1314.086,A -85,B 0,C 180,E1 991.444,E2 991.444} C_VEL
LIN {X 0,Y 599.994,Z 1309.75,A -85,B 0,C 180,E1 995.053,E2 995.053} C_VEL
LIN {X 0,Y 599.98,Z 1299.064,A -85,B 0,C 180,E1 999.047,E2 999.047} C_VEL
LIN {X 0,Y 600.044,Z 1283.436,A -85,B 0,C 180,E1 1002.715,E2 1002.715} C_VEL
LIN {X 0,Y 600.116,Z 1261.697,A -85,B 0,C 180,E1 1006.337,E2 1006.337} C_VEL
LIN {X 0,Y 600.355,Z 1236.031,A -85,B 0,C 180,E1 1009.545,E2 1009.545} C_VEL
LIN {X 0,Y 600.638,Z 1205.428,A -85,B 0,C 180,E1 1012.482,E2 1012.482} C_VEL
LIN {X 0,Y 600.999,Z 1170.85,A -85,B 0,C 180,E1 1015.005,E2 1015.005} C_VEL
LIN {X 0,Y 601.371,Z 1132.781,A -85,B 0,C 180,E1 1017.039,E2 1017.039} C_VEL
LIN {X 0,Y 601.584,Z 1093.373,A -85,B 0,C 180,E1 1018.467,E2 1018.467} C_VEL
LIN {X 0,Y 601.809,Z 1054.158,A -85,B 0,C 180,E1 1019.275,E2 1019.275} C_VEL
LIN {X 0,Y 600.771,Z 992.645,A -85,B 0,C 180,E1 1020.16,E2 1020.16} C_VEL
LIN {X 0,Y 599.933,Z 989.03,A -85,B 0,C 180,E1 1020.326,E2 1020.326} C_VEL
LIN {X 0,Y 599.661,Z 989.03,A -85,B 0,C 180,E1 1027.158,E2 1027.158} C_VEL
LIN {X 0,Y 599.574,Z 989.03,A -85,B 0,C 180,E1 1033.127,E2 1033.127} C_VEL
LIN {X 0,Y 599.41,Z 989.03,A -85,B 0,C 180,E1 1039.117,E2 1039.117} C_VEL
LIN {X 0,Y 599.303,Z 989.03,A -85,B 0,C 180,E1 1043.689,E2 1043.689} C_VEL
LIN {X 0,Y 599.605,Z 989.03,A -85,B 0,C 180,E1 1048.097,E2 1048.097} C_VEL
LIN {X 0,Y 599.479,Z 989.03,A -85,B 0,C 180,E1 1053.059,E2 1053.059} C_VEL
LIN {X 0,Y 599.553,Z 989.03,A -85,B 0,C 180,E1 1058.642,E2 1058.642} C_VEL
LIN {X 0,Y 599.794,Z 989.03,A -85,B 0,C 180,E1 1061.433,E2 1061.433} C_VEL
LIN {X 0,Y 600.613,Z 1031.21,A -85,B 0,C 180,E1 1062.17,E2 1062.17} C_VEL
LIN {X 0,Y 600.51,Z 1061.758,A -85,B 0,C 180,E1 1063.28,E2 1063.28} C_VEL
LIN {X 0,Y 600.358,Z 1090.74,A -85,B 0,C 180,E1 1064.974,E2 1064.974} C_VEL
LIN {X 0,Y 600.188,Z 1115.471,A -85,B 0,C 180,E1 1067.107,E2 1067.107} C_VEL
LIN {X 0,Y 600.017,Z 1135.546,A -85,B 0,C 180,E1 1069.584,E2 1069.584} C_VEL
LIN {X 0,Y 599.988,Z 1149.35,A -85,B 0,C 180,E1 1072.049,E2 1072.049} C_VEL
LIN {X 0,Y 599.926,Z 1159.512,A -85,B 0,C 180,E1 1074.949,E2 1074.949} C_VEL
LIN {X 0,Y 599.992,Z 1163.429,A -85,B 0,C 180,E1 1077.117,E2 1077.117} C_VEL
LIN {X 0,Y 599.984,Z 1164.128,A -85,B 0,C 180,E1 1080,E2 1080} C_VEL
LIN {X 0,Y 599.981,Z 1159.716,A -85,B 0,C 180,E1 1082.883,E2 1082.883} C_VEL
LIN {X 0,Y 600.043,Z 1149.761,A -85,B 0,C 180,E1 1085.773,E2 1085.773} C_VEL
LIN {X 0,Y 600.062,Z 1134.418,A -85,B 0,C 180,E1 1088.495,E2 1088.495} C_VEL
LIN {X 0,Y 600.212,Z 1113.329,A -85,B 0,C 180,E1 1091.024,E2 1091.024} C_VEL
LIN {X 0,Y 600.356,Z 1088.748,A -85,B 0,C 180,E1 1093.074,E2 1093.074} C_VEL
LIN {X 0,Y 600.528,Z 1060.974,A -85,B 0,C 180,E1 1094.667,E2 1094.667} C_VEL
LIN {X 0,Y 600.677,Z 1030.327,A -85,B 0,C 180,E1 1095.76,E2 1095.76} C_VEL
LIN {X 0,Y 599.605,Z 993.302,A -85,B 0,C 180,E1 1096.407,E2 1096.407} C_VEL
LIN {X 0,Y 599.475,Z 989.03,A -85,B 0,C 180,E1 1096.503,E2 1096.503} C_VEL
LIN {X 0,Y 599.616,Z 989.03,A -85,B 0,C 180,E1 1101.373,E2 1101.373} C_VEL
LIN {X 0,Y 599.609,Z 989.03,A -85,B 0,C 180,E1 1106.935,E2 1106.935} C_VEL
LIN {X 0,Y 599.728,Z 989.03,A -85,B 0,C 180,E1 1113.609,E2 1113.609} C_VEL
LIN {X 0,Y 599.582,Z 989.03,A -85,B 0,C 180,E1 1118.988,E2 1118.988} C_VEL
LIN {X 0,Y 599.548,Z 989.03,A -85,B 0,C 180,E1 1125.186,E2 1125.186} C_VEL
LIN {X 0,Y 599.536,Z 989.03,A -85,B 0,C 180,E1 1131.001,E2 1131.001} C_VEL
LIN {X 0,Y 599.563,Z 989.03,A -85,B 0,C 180,E1 1134.624,E2 1134.624} C_VEL
LIN {X 0,Y 599.624,Z 989.03,A -85,B 0,C 180,E1 1139.776,E2 1139.776} C_VEL
LIN {X 0,Y 599.37,Z 989.03,A -85,B 0,C 180,E1 1144.22,E2 1144.22} C_VEL
LIN {X 0,Y 601.166,Z 998.596,A -85,B 0,C 180,E1 1144.446,E2 1144.446} C_VEL
LIN {X 0,Y 601.244,Z 1043.615,A -85,B 0,C 180,E1 1145.179,E2 1145.179} C_VEL
LIN {X 0,Y 601.107,Z 1079.237,A -85,B 0,C 180,E1 1146.314,E2 1146.314} C_VEL
LIN {X 0,Y 600.797,Z 1112.998,A -85,B 0,C 180,E1 1147.953,E2 1147.953} C_VEL
LIN {X 0,Y 600.571,Z 1145.669,A -85,B 0,C 180,E1 1150.172,E2 1150.172} C_VEL
LIN {X 0,Y 600.245,Z 1174.268,A -85,B 0,C 180,E1 1152.798,E2 1152.798} C_VEL
LIN {X 0,Y 600.046,Z 1198.794,A -85,B 0,C 180,E1 1155.804,E2 1155.804} C_VEL
LIN {X 0,Y 599.921,Z 1217.706,A -85,B 0,C 180,E1 1158.945,E2 1158.945} C_VEL
LIN {X 0,Y 599.867,Z 1232.171,A -85,B 0,C 180,E1 1162.408,E2 1162.408} C_VEL
LIN {X 0,Y 599.835,Z 1240.564,A -85,B 0,C 180,E1 1165.669,E2 1165.669} C_VEL
LIN {X 0,Y 599.872,Z 1244.04,A -85,B 0,C 180,E1 1168.556,E2 1168.556} C_VEL
LIN {X 0,Y 599.996,Z 1243.981,A -85,B 0,C 180,E1 1171.438,E2 1171.438} C_VEL
LIN {X 0,Y 599.934,Z 1238.897,A -85,B 0,C 180,E1 1175.048,E2 1175.048} C_VEL
LIN {X 0,Y 599.96,Z 1227.95,A -85,B 0,C 180,E1 1178.677,E2 1178.677} C_VEL
LIN {X 0,Y 600.034,Z 1211.206,A -85,B 0,C 180,E1 1182.156,E2 1182.156} C_VEL
LIN {X 0,Y 600.162,Z 1189.844,A -85,B 0,C 180,E1 1185.305,E2 1185.305} C_VEL
LIN {X 0,Y 600.393,Z 1163.295,A -85,B 0,C 180,E1 1188.214,E2 1188.214} C_VEL
LIN {X 0,Y 600.688,Z 1132.36,A -85,B 0,C 180,E1 1190.724,E2 1190.724} C_VEL
LIN {X 0,Y 600.937,Z 1098.876,A -85,B 0,C 180,E1 1192.718,E2 1192.718} C_VEL
LIN {X 0,Y 601.208,Z 1063.62,A -85,B 0,C 180,E1 1194.167,E2 1194.167} C_VEL
LIN {X 0,Y 601.39,Z 1027.161,A -85,B 0,C 180,E1 1195.062,E2 1195.062} C_VEL
LIN {X 0,Y 600.51,Z 991.84,A -85,B 0,C 180,E1 1195.582,E2 1195.582} C_VEL
LIN {X 0,Y 599.958,Z 989.03,A -85,B 0,C 180,E1 1195.66,E2 1195.66} C_VEL
LIN {X 0,Y 599.389,Z 989.03,A -85,B 0,C 180,E1 1201.137,E2 1201.137} C_VEL
LIN {X 0,Y 599.393,Z 989.03,A -85,B 0,C 180,E1 1205.381,E2 1205.381} C_VEL
LIN {X 0,Y 599.614,Z 989.03,A -85,B 0,C 180,E1 1208.986,E2 1208.986} C_VEL
LIN {X 0,Y 599.529,Z 989.03,A -85,B 0,C 180,E1 1215.193,E2 1215.193} C_VEL
LIN {X 0,Y 599.527,Z 989.03,A -85,B 0,C 180,E1 1221.008,E2 1221.008} C_VEL
LIN {X 0,Y 599.566,Z 989.03,A -85,B 0,C 180,E1 1224.631,E2 1224.631} C_VEL
LIN {X 0,Y 599.63,Z 989.03,A -85,B 0,C 180,E1 1229.782,E2 1229.782} C_VEL
LIN {X 0,Y 599.867,Z 989.03,A -85,B 0,C 180,E1 1234.902,E2 1234.902} C_VEL
LIN {X 0,Y 599.778,Z 989.03,A -85,B 0,C 180,E1 1240.91,E2 1240.91} C_VEL
LIN {X 0,Y 599.965,Z 989.03,A -85,B 0,C 180,E1 1246.918,E2 1246.918} C_VEL
LIN {X 0,Y 599.722,Z 989.03,A -85,B 0,C 180,E1 1252.773,E2 1252.773} C_VEL
LIN {X 0,Y 599.838,Z 989.03,A -85,B 0,C 180,E1 1257.116,E2 1257.116} C_VEL
LIN {X 0,Y 599.577,Z 989.03,A -85,B 0,C 180,E1 1259.146,E2 1259.146} C_VEL
LIN {X 0,Y 598.41,Z 989.03,A -85,B 0,C 180,E1 1259.975,E2 1259.975} C_VEL
LIN {X 0,Y 591.787,Z 989.03,A -85,B 0,C 180,E1 1262.442,E2 1262.442} C_VEL
LIN {X 0,Y 591.701,Z 989.03,A -85,B 0,C 180,E1 1267.326,E2 1267.326} C_VEL
LIN {X 0,Y 591.732,Z 989.03,A -85,B 0,C 180,E1 1271.771,E2 1271.771} C_VEL
LIN {X 0,Y 591.759,Z 989.03,A -85,B 0,C 180,E1 1276.29,E2 1276.29} C_VEL
LIN {X 0,Y 591.797,Z 989.03,A -85,B 0,C 180,E1 1280.914,E2 1280.914} C_VEL
LIN {X 0,Y 591.634,Z 989.03,A -85,B 0,C 180,E1 1286.788,E2 1286.788} C_VEL
LIN {X 0,Y 591.665,Z 989.03,A -85,B 0,C 180,E1 1290.668,E2 1290.668} C_VEL
LIN {X 0,Y 591.728,Z 989.03,A -85,B 0,C 180,E1 1295.91,E2 1295.91} C_VEL
LIN {X 0,Y 591.646,Z 989.03,A -85,B 0,C 180,E1 1301.538,E2 1301.538} C_VEL
LIN {X 0,Y 591.505,Z 989.03,A -85,B 0,C 180,E1 1306.467,E2 1306.467} C_VEL
LIN {X 0,Y 591.536,Z 989.03,A -85,B 0,C 180,E1 1312.258,E2 1312.258} C_VEL
LIN {X 0,Y 591.818,Z 989.03,A -85,B 0,C 180,E1 1317.627,E2 1317.627} C_VEL
LIN {X 0,Y 591.974,Z 989.43,A -85,B 0,C 180,E1 1319.299,E2 1319.299} C_VEL
LIN {X 0,Y 594.649,Z 999.09,A -85,B 0,C 180,E1 1319.585,E2 1319.585} C_VEL
LIN {X 0,Y 594.68,Z 1077.386,A -85,B 0,C 180,E1 1320.763,E2 1320.763} C_VEL
LIN {X 0,Y 594.404,Z 1114.348,A -85,B 0,C 180,E1 1321.858,E2 1321.858} C_VEL
LIN {X 0,Y 593.955,Z 1150.865,A -85,B 0,C 180,E1 1323.502,E2 1323.502} C_VEL
LIN {X 0,Y 593.411,Z 1186.321,A -85,B 0,C 180,E1 1325.719,E2 1325.719} C_VEL
LIN {X 0,Y 592.952,Z 1219.394,A -85,B 0,C 180,E1 1328.475,E2 1328.475} C_VEL
LIN {X 0,Y 592.531,Z 1248.309,A -85,B 0,C 180,E1 1331.632,E2 1331.632} C_VEL
LIN {X 0,Y 592.195,Z 1272.081,A -85,B 0,C 180,E1 1335.051,E2 1335.051} C_VEL
LIN {X 0,Y 592,Z 1290.066,A -85,B 0,C 180,E1 1338.518,E2 1338.518} C_VEL
LIN {X 0,Y 591.972,Z 1303.723,A -85,B 0,C 180,E1 1342.312,E2 1342.312} C_VEL
LIN {X 0,Y 591.872,Z 1310.966,A -85,B 0,C 180,E1 1345.616,E2 1345.616} C_VEL
LIN {X 0,Y 591.9,Z 1314.092,A -85,B 0,C 180,E1 1348.542,E2 1348.542} C_VEL
LIN {X 0,Y 592.073,Z 1314.088,A -85,B 0,C 180,E1 1351.463,E2 1351.463} C_VEL
LIN {X 0,Y 592.093,Z 1309.748,A -85,B 0,C 180,E1 1355.121,E2 1355.121} C_VEL
LIN {X 0,Y 592.096,Z 1299.066,A -85,B 0,C 180,E1 1359.169,E2 1359.169} C_VEL
LIN {X 0,Y 592.192,Z 1283.438,A -85,B 0,C 180,E1 1362.887,E2 1362.887} C_VEL
LIN {X 0,Y 592.352,Z 1261.932,A -85,B 0,C 180,E1 1366.524,E2 1366.524} C_VEL
LIN {X 0,Y 592.671,Z 1235.966,A -85,B 0,C 180,E1 1369.816,E2 1369.816} C_VEL
LIN {X 0,Y 593.119,Z 1205.727,A -85,B 0,C 180,E1 1372.758,E2 1372.758} C_VEL
LIN {X 0,Y 593.659,Z 1171.633,A -85,B 0,C 180,E1 1375.284,E2 1375.284} C_VEL
LIN {X 0,Y 594.207,Z 1133.885,A -85,B 0,C 180,E1 1377.341,E2 1377.341} C_VEL
LIN {X 0,Y 594.593,Z 1094.6,A -85,B 0,C 180,E1 1378.798,E2 1378.798} C_VEL
LIN {X 0,Y 594.927,Z 1056.585,A -85,B 0,C 180,E1 1379.61,E2 1379.61} C_VEL
LIN {X 0,Y 594.191,Z 995.527,A -85,B 0,C 180,E1 1380.49,E2 1380.49} C_VEL
LIN {X 0,Y 591.978,Z 989.03,A -85,B 0,C 180,E1 1380.707,E2 1380.707} C_VEL
LIN {X 0,Y 591.695,Z 989.03,A -85,B 0,C 180,E1 1385.919,E2 1385.919} C_VEL
LIN {X 0,Y 591.646,Z 989.03,A -85,B 0,C 180,E1 1391.545,E2 1391.545} C_VEL
LIN {X 0,Y 591.505,Z 989.03,A -85,B 0,C 180,E1 1396.467,E2 1396.467} C_VEL
LIN {X 0,Y 591.534,Z 989.03,A -85,B 0,C 180,E1 1402.268,E2 1402.268} C_VEL
LIN {X 0,Y 591.693,Z 989.03,A -85,B 0,C 180,E1 1407.619,E2 1407.619} C_VEL
LIN {X 0,Y 591.585,Z 989.03,A -85,B 0,C 180,E1 1413.234,E2 1413.234} C_VEL
LIN {X 0,Y 591.685,Z 989.03,A -85,B 0,C 180,E1 1417.509,E2 1417.509} C_VEL
LIN {X 0,Y 591.988,Z 989.03,A -85,B 0,C 180,E1 1421.179,E2 1421.179} C_VEL
LIN {X 0,Y 593.121,Z 1012.262,A -85,B 0,C 180,E1 1421.553,E2 1421.553} C_VEL
LIN {X 0,Y 593,Z 1044.03,A -85,B 0,C 180,E1 1422.348,E2 1422.348} C_VEL
LIN {X 0,Y 592.785,Z 1073.284,A -85,B 0,C 180,E1 1423.672,E2 1423.672} C_VEL
LIN {X 0,Y 592.549,Z 1100.776,A -85,B 0,C 180,E1 1425.574,E2 1425.574} C_VEL
LIN {X 0,Y 592.337,Z 1123.713,A -85,B 0,C 180,E1 1427.868,E2 1427.868} C_VEL
LIN {X 0,Y 592.235,Z 1141.737,A -85,B 0,C 180,E1 1430.467,E2 1430.467} C_VEL
LIN {X 0,Y 592.143,Z 1154.732,A -85,B 0,C 180,E1 1433.303,E2 1433.303} C_VEL
LIN {X 0,Y 592.178,Z 1162.424,A -85,B 0,C 180,E1 1436.347,E2 1436.347} C_VEL
LIN {X 0,Y 592.045,Z 1164.415,A -85,B 0,C 180,E1 1438.539,E2 1438.539} C_VEL
LIN {X 0,Y 592.092,Z 1162.591,A -85,B 0,C 180,E1 1441.46,E2 1441.46} C_VEL
LIN {X 0,Y 592.117,Z 1155.526,A -85,B 0,C 180,E1 1444.384,E2 1444.384} C_VEL
LIN {X 0,Y 592.196,Z 1142.466,A -85,B 0,C 180,E1 1447.319,E2 1447.319} C_VEL
LIN {X 0,Y 592.35,Z 1124.86,A -85,B 0,C 180,E1 1449.901,E2 1449.901} C_VEL
LIN {X 0,Y 592.536,Z 1102.176,A -85,B 0,C 180,E1 1452.221,E2 1452.221} C_VEL
LIN {X 0,Y 592.727,Z 1075.73,A -85,B 0,C 180,E1 1454.099,E2 1454.099} C_VEL
LIN {X 0,Y 592.971,Z 1045.95,A -85,B 0,C 180,E1 1455.497,E2 1455.497} C_VEL
LIN {X 0,Y 593.055,Z 1013.704,A -85,B 0,C 180,E1 1456.336,E2 1456.336} C_VEL
LIN {X 0,Y 591.806,Z 989.03,A -85,B 0,C 180,E1 1456.734,E2 1456.734} C_VEL
LIN {X 0,Y 591.75,Z 989.03,A -85,B 0,C 180,E1 1462.488,E2 1462.488} C_VEL
LIN {X 0,Y 591.734,Z 989.03,A -85,B 0,C 180,E1 1467.323,E2 1467.323} C_VEL
LIN {X 0,Y 591.726,Z 989.03,A -85,B 0,C 180,E1 1474.126,E2 1474.126} C_VEL
LIN {X 0,Y 591.516,Z 989.03,A -85,B 0,C 180,E1 1480.058,E2 1480.058} C_VEL
LIN {X 0,Y 591.607,Z 989.03,A -85,B 0,C 180,E1 1485.574,E2 1485.574} C_VEL
LIN {X 0,Y 591.58,Z 989.03,A -85,B 0,C 180,E1 1490.374,E2 1490.374} C_VEL
LIN {X 0,Y 591.495,Z 989.03,A -85,B 0,C 180,E1 1495.852,E2 1495.852} C_VEL
LIN {X 0,Y 591.573,Z 989.03,A -85,B 0,C 180,E1 1501.006,E2 1501.006} C_VEL
LIN {X 0,Y 591.485,Z 989.452,A -85,B 0,C 180,E1 1503.877,E2 1503.877} C_VEL
LIN {X 0,Y 594.029,Z 998.58,A -85,B 0,C 180,E1 1504.117,E2 1504.117} C_VEL
LIN {X 0,Y 594.028,Z 1043.605,A -85,B 0,C 180,E1 1504.857,E2 1504.857} C_VEL
LIN {X 0,Y 593.837,Z 1079.229,A -85,B 0,C 180,E1 1506.006,E2 1506.006} C_VEL
LIN {X 0,Y 593.355,Z 1113.464,A -85,B 0,C 180,E1 1507.689,E2 1507.689} C_VEL
LIN {X 0,Y 592.984,Z 1146.655,A -85,B 0,C 180,E1 1509.986,E2 1509.986} C_VEL
LIN {X 0,Y 592.519,Z 1175.601,A -85,B 0,C 180,E1 1512.712,E2 1512.712} C_VEL
LIN {X 0,Y 592.251,Z 1200.116,A -85,B 0,C 180,E1 1515.802,E2 1515.802} C_VEL
LIN {X 0,Y 592.068,Z 1218.841,A -85,B 0,C 180,E1 1519.028,E2 1519.028} C_VEL
LIN {X 0,Y 591.984,Z 1232.17,A -85,B 0,C 180,E1 1522.306,E2 1522.306} C_VEL
LIN {X 0,Y 591.939,Z 1240.563,A -85,B 0,C 180,E1 1525.611,E2 1525.611} C_VEL
LIN {X 0,Y 591.972,Z 1244.04,A -85,B 0,C 180,E1 1528.536,E2 1528.536} C_VEL
LIN {X 0,Y 592.092,Z 1243.982,A -85,B 0,C 180,E1 1531.458,E2 1531.458} C_VEL
LIN {X 0,Y 592.036,Z 1238.899,A -85,B 0,C 180,E1 1535.115,E2 1535.115} C_VEL
LIN {X 0,Y 592.088,Z 1227.953,A -85,B 0,C 180,E1 1538.793,E2 1538.793} C_VEL
LIN {X 0,Y 592.162,Z 1211.213,A -85,B 0,C 180,E1 1542.32,E2 1542.32} C_VEL
LIN {X 0,Y 592.372,Z 1189.852,A -85,B 0,C 180,E1 1545.512,E2 1545.512} C_VEL
LIN {X 0,Y 592.717,Z 1163.299,A -85,B 0,C 180,E1 1548.458,E2 1548.458} C_VEL
LIN {X 0,Y 593.136,Z 1132.709,A -85,B 0,C 180,E1 1550.976,E2 1550.976} C_VEL
LIN {X 0,Y 593.582,Z 1098.825,A -85,B 0,C 180,E1 1553.019,E2 1553.019} C_VEL
LIN {X 0,Y 593.986,Z 1062.685,A -85,B 0,C 180,E1 1554.51,E2 1554.51} C_VEL
LIN {X 0,Y 594.229,Z 1027.178,A -85,B 0,C 180,E1 1555.386,E2 1555.386} C_VEL
LIN {X 0,Y 593.618,Z 994.322,A -85,B 0,C 180,E1 1555.869,E2 1555.869} C_VEL
LIN {X 0,Y 592.052,Z 989.03,A -85,B 0,C 180,E1 1556.043,E2 1556.043} C_VEL
LIN {X 0,Y 591.67,Z 989.03,A -85,B 0,C 180,E1 1562.691,E2 1562.691} C_VEL
LIN {X 0,Y 591.531,Z 989.03,A -85,B 0,C 180,E1 1567.75,E2 1567.75} C_VEL
LIN {X 0,Y 591.53,Z 989.03,A -85,B 0,C 180,E1 1573.531,E2 1573.531} C_VEL
LIN {X 0,Y 591.64,Z 989.03,A -85,B 0,C 180,E1 1578.463,E2 1578.463} C_VEL
LIN {X 0,Y 591.725,Z 989.03,A -85,B 0,C 180,E1 1584.09,E2 1584.09} C_VEL
LIN {X 0,Y 591.659,Z 989.03,A -85,B 0,C 180,E1 1590.128,E2 1590.128} C_VEL
LIN {X 0,Y 591.671,Z 989.03,A -85,B 0,C 180,E1 1595.918,E2 1595.918} C_VEL
LIN {X 0,Y 591.878,Z 989.03,A -85,B 0,C 180,E1 1600.645,E2 1600.645} C_VEL
LIN {X 0,Y 592.02,Z 989.03,A -85,B 0,C 180,E1 1606.739,E2 1606.739} C_VEL
LIN {X 0,Y 591.83,Z 989.03,A -85,B 0,C 180,E1 1612.702,E2 1612.702} C_VEL
LIN {X 0,Y 591.932,Z 989.03,A -85,B 0,C 180,E1 1617.078,E2 1617.078} C_VEL
LIN {X 0,Y 591.787,Z 989.03,A -85,B 0,C 180,E1 1622.442,E2 1622.442} C_VEL
LIN {X 0,Y 587.747,Z 989.03,A -85,B 0,C 180,E1 1624.1,E2 1624.1} C_VEL
LIN {X 0,Y 584.103,Z 989.03,A -85,B 0,C 180,E1 1625.779,E2 1625.779} C_VEL
LIN {X 0,Y 583.814,Z 989.03,A -85,B 0,C 180,E1 1631.933,E2 1631.933} C_VEL
LIN {X 0,Y 583.739,Z 989.03,A -85,B 0,C 180,E1 1636.97,E2 1636.97} C_VEL
LIN {X 0,Y 583.751,Z 989.03,A -85,B 0,C 180,E1 1641.474,E2 1641.474} C_VEL
LIN {X 0,Y 583.823,Z 989.03,A -85,B 0,C 180,E1 1646.065,E2 1646.065} C_VEL
LIN {X 0,Y 583.604,Z 989.03,A -85,B 0,C 180,E1 1651.433,E2 1651.433} C_VEL
LIN {X 0,Y 583.759,Z 989.03,A -85,B 0,C 180,E1 1656.744,E2 1656.744} C_VEL
LIN {X 0,Y 583.743,Z 989.03,A -85,B 0,C 180,E1 1662.228,E2 1662.228} C_VEL
LIN {X 0,Y 583.544,Z 989.03,A -85,B 0,C 180,E1 1667.754,E2 1667.754} C_VEL
LIN {X 0,Y 583.518,Z 989.03,A -85,B 0,C 180,E1 1673.287,E2 1673.287} C_VEL
LIN {X 0,Y 584.01,Z 989.166,A -85,B 0,C 180,E1 1678.831,E2 1678.831} C_VEL
LIN {X 0,Y 587.773,Z 998.869,A -85,B 0,C 180,E1 1679.187,E2 1679.187} C_VEL
LIN {X 0,Y 587.767,Z 1078.981,A -85,B 0,C 180,E1 1680.42,E2 1680.42} C_VEL
LIN {X 0,Y 587.349,Z 1116.643,A -85,B 0,C 180,E1 1681.576,E2 1681.576} C_VEL
LIN {X 0,Y 586.709,Z 1152.833,A -85,B 0,C 180,E1 1683.257,E2 1683.257} C_VEL
LIN {X 0,Y 585.991,Z 1187.665,A -85,B 0,C 180,E1 1685.491,E2 1685.491} C_VEL
LIN {X 0,Y 585.372,Z 1220.477,A -85,B 0,C 180,E1 1688.285,E2 1688.285} C_VEL
LIN {X 0,Y 584.789,Z 1249.804,A -85,B 0,C 180,E1 1691.575,E2 1691.575} C_VEL
LIN {X 0,Y 584.375,Z 1273.172,A -85,B 0,C 180,E1 1695.038,E2 1695.038} C_VEL
LIN {X 0,Y 584.15,Z 1291.048,A -85,B 0,C 180,E1 1698.598,E2 1698.598} C_VEL
LIN {X 0,Y 584.097,Z 1303.722,A -85,B 0,C 180,E1 1702.207,E2 1702.207} C_VEL
LIN {X 0,Y 583.985,Z 1310.969,A -85,B 0,C 180,E1 1705.557,E2 1705.557} C_VEL
LIN {X 0,Y 584.026,Z 1314.094,A -85,B 0,C 180,E1 1708.522,E2 1708.522} C_VEL
LIN {X 0,Y 584.183,Z 1314.09,A -85,B 0,C 180,E1 1711.483,E2 1711.483} C_VEL
LIN {X 0,Y 584.21,Z 1309.744,A -85,B 0,C 180,E1 1715.19,E2 1715.19} C_VEL
LIN {X 0,Y 584.19,Z 1299.068,A -85,B 0,C 180,E1 1719.294,E2 1719.294} C_VEL
LIN {X 0,Y 584.331,Z 1283.433,A -85,B 0,C 180,E1 1723.063,E2 1723.063} C_VEL
LIN {X 0,Y 584.558,Z 1262.362,A -85,B 0,C 180,E1 1726.689,E2 1726.689} C_VEL
LIN {X 0,Y 585.021,Z 1236.752,A -85,B 0,C 180,E1 1729.998,E2 1729.998} C_VEL
LIN {X 0,Y 585.614,Z 1206.247,A -85,B 0,C 180,E1 1733.021,E2 1733.021} C_VEL
LIN {X 0,Y 586.322,Z 1172.614,A -85,B 0,C 180,E1 1735.557,E2 1735.557} C_VEL
LIN {X 0,Y 587.027,Z 1136.682,A -85,B 0,C 180,E1 1737.566,E2 1737.566} C_VEL
LIN {X 0,Y 587.58,Z 1099.344,A -85,B 0,C 180,E1 1739.022,E2 1739.022} C_VEL
LIN {X 0,Y 588.012,Z 1064.519,A -85,B 0,C 180,E1 1739.864,E2 1739.864} C_VEL
LIN {X 0,Y 587.368,Z 997.657,A -85,B 0,C 180,E1 1740.853,E2 1740.853} C_VEL
LIN {X 0,Y 583.879,Z 989.03,A -85,B 0,C 180,E1 1741.181,E2 1741.181} C_VEL
LIN {X 0,Y 583.743,Z 989.03,A -85,B 0,C 180,E1 1746.742,E2 1746.742} C_VEL
LIN {X 0,Y 583.745,Z 989.03,A -85,B 0,C 180,E1 1752.236,E2 1752.236} C_VEL
LIN {X 0,Y 583.543,Z 989.03,A -85,B 0,C 180,E1 1757.754,E2 1757.754} C_VEL
LIN {X 0,Y 583.508,Z 989.03,A -85,B 0,C 180,E1 1763.299,E2 1763.299} C_VEL
LIN {X 0,Y 583.837,Z 989.03,A -85,B 0,C 180,E1 1767.129,E2 1767.129} C_VEL
LIN {X 0,Y 583.694,Z 989.03,A -85,B 0,C 180,E1 1772.268,E2 1772.268} C_VEL
LIN {X 0,Y 583.799,Z 989.03,A -85,B 0,C 180,E1 1777.188,E2 1777.188} C_VEL
LIN {X 0,Y 584.046,Z 989.03,A -85,B 0,C 180,E1 1780.963,E2 1780.963} C_VEL
LIN {X 0,Y 585.586,Z 1007.242,A -85,B 0,C 180,E1 1781.247,E2 1781.247} C_VEL
LIN {X 0,Y 585.417,Z 1039.804,A -85,B 0,C 180,E1 1781.982,E2 1781.982} C_VEL
LIN {X 0,Y 585.166,Z 1069.938,A -85,B 0,C 180,E1 1783.277,E2 1783.277} C_VEL
LIN {X 0,Y 584.832,Z 1097.666,A -85,B 0,C 180,E1 1785.136,E2 1785.136} C_VEL
LIN {X 0,Y 584.502,Z 1120.385,A -85,B 0,C 180,E1 1787.324,E2 1787.324} C_VEL
LIN {X 0,Y 584.326,Z 1139.472,A -85,B 0,C 180,E1 1789.961,E2 1789.961} C_VEL
LIN {X 0,Y 584.215,Z 1152.336,A -85,B 0,C 180,E1 1792.58,E2 1792.58} C_VEL
LIN {X 0,Y 584.175,Z 1161.095,A -85,B 0,C 180,E1 1795.555,E2 1795.555} C_VEL
LIN {X 0,Y 584.165,Z 1164.413,A -85,B 0,C 180,E1 1798.52,E2 1798.52} C_VEL
LIN {X 0,Y 584.211,Z 1162.609,A -85,B 0,C 180,E1 1801.48,E2 1801.48} C_VEL
LIN {X 0,Y 584.234,Z 1155.568,A -85,B 0,C 180,E1 1804.444,E2 1804.444} C_VEL
LIN {X 0,Y 584.333,Z 1142.543,A -85,B 0,C 180,E1 1807.418,E2 1807.418} C_VEL
LIN {X 0,Y 584.548,Z 1123.461,A -85,B 0,C 180,E1 1810.222,E2 1810.222} C_VEL
LIN {X 0,Y 584.783,Z 1100.084,A -85,B 0,C 180,E1 1812.575,E2 1812.575} C_VEL
LIN {X 0,Y 585.114,Z 1073.114,A -85,B 0,C 180,E1 1814.453,E2 1814.453} C_VEL
LIN {X 0,Y 585.447,Z 1043.612,A -85,B 0,C 180,E1 1815.797,E2 1815.797} C_VEL
LIN {X 0,Y 585.484,Z 1011.797,A -85,B 0,C 180,E1 1816.598,E2 1816.598} C_VEL
LIN {X 0,Y 583.987,Z 989.03,A -85,B 0,C 180,E1 1816.968,E2 1816.968} C_VEL
LIN {X 0,Y 583.847,Z 989.03,A -85,B 0,C 180,E1 1822.809,E2 1822.809} C_VEL
LIN {X 0,Y 583.704,Z 989.03,A -85,B 0,C 180,E1 1828.472,E2 1828.472} C_VEL
LIN {X 0,Y 583.733,Z 989.03,A -85,B 0,C 180,E1 1834.659,E2 1834.659} C_VEL
LIN {X 0,Y 583.583,Z 989.03,A -85,B 0,C 180,E1 1840.271,E2 1840.271} C_VEL
LIN {X 0,Y 583.715,Z 989.03,A -85,B 0,C 180,E1 1845.728,E2 1845.728} C_VEL
LIN {X 0,Y 583.724,Z 989.03,A -85,B 0,C 180,E1 1851.647,E2 1851.647} C_VEL
LIN {X 0,Y 583.528,Z 989.03,A -85,B 0,C 180,E1 1857.103,E2 1857.103} C_VEL
LIN {X 0,Y 583.522,Z 989.03,A -85,B 0,C 180,E1 1862.254,E2 1862.254} C_VEL
LIN {X 0,Y 583.542,Z 989.03,A -85,B 0,C 180,E1 1863.467,E2 1863.467} C_VEL
LIN {X 0,Y 586.922,Z 999.485,A -85,B 0,C 180,E1 1863.792,E2 1863.792} C_VEL
LIN {X 0,Y 586.85,Z 1044.951,A -85,B 0,C 180,E1 1864.563,E2 1864.563} C_VEL
LIN {X 0,Y 586.553,Z 1080.303,A -85,B 0,C 180,E1 1865.735,E2 1865.735} C_VEL
LIN {X 0,Y 585.918,Z 1114.718,A -85,B 0,C 180,E1 1867.465,E2 1867.465} C_VEL
LIN {X 0,Y 585.397,Z 1146.973,A -85,B 0,C 180,E1 1869.743,E2 1869.743} C_VEL
LIN {X 0,Y 584.792,Z 1176.277,A -85,B 0,C 180,E1 1872.552,E2 1872.552} C_VEL
LIN {X 0,Y 584.442,Z 1200.847,A -85,B 0,C 180,E1 1875.717,E2 1875.717} C_VEL
LIN {X 0,Y 584.21,Z 1219.937,A -85,B 0,C 180,E1 1879.116,E2 1879.116} C_VEL
LIN {X 0,Y 584.109,Z 1233.311,A -85,B 0,C 180,E1 1882.575,E2 1882.575} C_VEL
LIN {X 0,Y 584.054,Z 1240.562,A -85,B 0,C 180,E1 1885.552,E2 1885.552} C_VEL
LIN {X 0,Y 584.093,Z 1244.04,A -85,B 0,C 180,E1 1888.517,E2 1888.517} C_VEL
LIN {X 0,Y 584.203,Z 1243.982,A -85,B 0,C 180,E1 1891.477,E2 1891.477} C_VEL
LIN {X 0,Y 584.156,Z 1238.9,A -85,B 0,C 180,E1 1895.185,E2 1895.185} C_VEL
LIN {X 0,Y 584.19,Z 1227.957,A -85,B 0,C 180,E1 1898.913,E2 1898.913} C_VEL
LIN {X 0,Y 584.316,Z 1212.294,A -85,B 0,C 180,E1 1902.299,E2 1902.299} C_VEL
LIN {X 0,Y 584.602,Z 1191.323,A -85,B 0,C 180,E1 1905.531,E2 1905.531} C_VEL
LIN {X 0,Y 585.027,Z 1166.216,A -85,B 0,C 180,E1 1908.417,E2 1908.417} C_VEL
LIN {X 0,Y 585.592,Z 1135.672,A -85,B 0,C 180,E1 1911.046,E2 1911.046} C_VEL
LIN {X 0,Y 586.132,Z 1103.411,A -85,B 0,C 180,E1 1913.085,E2 1913.085} C_VEL
LIN {X 0,Y 586.66,Z 1068.454,A -85,B 0,C 180,E1 1914.634,E2 1914.634} C_VEL
LIN {X 0,Y 587.061,Z 1031.693,A -85,B 0,C 180,E1 1915.636,E2 1915.636} C_VEL
LIN {X 0,Y 586.585,Z 996.623,A -85,B 0,C 180,E1 1916.172,E2 1916.172} C_VEL
LIN {X 0,Y 584.114,Z 989.03,A -85,B 0,C 180,E1 1916.464,E2 1916.464} C_VEL
LIN {X 0,Y 583.777,Z 989.03,A -85,B 0,C 180,E1 1922.874,E2 1922.874} C_VEL
LIN {X 0,Y 583.597,Z 989.03,A -85,B 0,C 180,E1 1929.134,E2 1929.134} C_VEL
LIN {X 0,Y 583.661,Z 989.03,A -85,B 0,C 180,E1 1934.27,E2 1934.27} C_VEL
LIN {X 0,Y 583.68,Z 989.03,A -85,B 0,C 180,E1 1939.737,E2 1939.737} C_VEL
LIN {X 0,Y 583.636,Z 989.03,A -85,B 0,C 180,E1 1945.334,E2 1945.334} C_VEL
LIN {X 0,Y 583.7,Z 989.03,A -85,B 0,C 180,E1 1950.583,E2 1950.583} C_VEL
LIN {X 0,Y 583.757,Z 989.03,A -85,B 0,C 180,E1 1955.57,E2 1955.57} C_VEL
LIN {X 0,Y 583.957,Z 989.03,A -85,B 0,C 180,E1 1960.372,E2 1960.372} C_VEL
LIN {X 0,Y 584.101,Z 989.03,A -85,B 0,C 180,E1 1966.556,E2 1966.556} C_VEL
LIN {X 0,Y 583.906,Z 989.03,A -85,B 0,C 180,E1 1972.686,E2 1972.686} C_VEL
LIN {X 0,Y 584.048,Z 989.03,A -85,B 0,C 180,E1 1977.038,E2 1977.038} C_VEL
LIN {X 0,Y 583.904,Z 989.03,A -85,B 0,C 180,E1 1982.429,E2 1982.429} C_VEL
LIN {X 0,Y 584.103,Z 989.03,A -85,B 0,C 180,E1 1985.779,E2 1985.779} C_VEL
LIN {X 0,Y 581.644,Z 989.03,A -85,B 0,C 180,E1 1987.04,E2 1987.04} C_VEL
LIN {X 0,Y 575.994,Z 989.03,A -85,B 0,C 180,E1 1988.924,E2 1988.924} C_VEL
LIN {X 0,Y 575.893,Z 989.03,A -85,B 0,C 180,E1 1989.143,E2 1989.143} C_VEL
LIN {X 0,Y 575.949,Z 989.03,A -85,B 0,C 180,E1 1995.189,E2 1995.189} C_VEL
LIN {X 0,Y 575.858,Z 989.03,A -85,B 0,C 180,E1 2001.522,E2 2001.522} C_VEL
LIN {X 0,Y 575.792,Z 989.03,A -85,B 0,C 180,E1 2006.997,E2 2006.997} C_VEL
LIN {X 0,Y 575.694,Z 989.03,A -85,B 0,C 180,E1 2011.616,E2 2011.616} C_VEL
LIN {X 0,Y 575.84,Z 989.03,A -85,B 0,C 180,E1 2017.064,E2 2017.064} C_VEL
LIN {X 0,Y 575.798,Z 989.03,A -85,B 0,C 180,E1 2022.95,E2 2022.95} C_VEL
LIN {X 0,Y 575.688,Z 989.03,A -85,B 0,C 180,E1 2029.475,E2 2029.475} C_VEL
LIN {X 0,Y 575.709,Z 989.03,A -85,B 0,C 180,E1 2034.787,E2 2034.787} C_VEL
LIN {X 0,Y 576.071,Z 989.176,A -85,B 0,C 180,E1 2038.352,E2 2038.352} C_VEL
LIN {X 0,Y 581.073,Z 1003.429,A -85,B 0,C 180,E1 2038.857,E2 2038.857} C_VEL
LIN {X 0,Y 580.913,Z 1077.519,A -85,B 0,C 180,E1 2040.002,E2 2040.002} C_VEL
LIN {X 0,Y 580.386,Z 1115.025,A -85,B 0,C 180,E1 2041.141,E2 2041.141} C_VEL
LIN {X 0,Y 579.61,Z 1150.941,A -85,B 0,C 180,E1 2042.797,E2 2042.797} C_VEL
LIN {X 0,Y 578.692,Z 1185.924,A -85,B 0,C 180,E1 2045.03,E2 2045.03} C_VEL
LIN {X 0,Y 577.83,Z 1218.766,A -85,B 0,C 180,E1 2047.821,E2 2047.821} C_VEL
LIN {X 0,Y 577.057,Z 1248.562,A -85,B 0,C 180,E1 2051.155,E2 2051.155} C_VEL
LIN {X 0,Y 576.535,Z 1272.079,A -85,B 0,C 180,E1 2054.635,E2 2054.635} C_VEL
LIN {X 0,Y 576.278,Z 1290.772,A -85,B 0,C 180,E1 2058.37,E2 2058.37} C_VEL
LIN {X 0,Y 576.202,Z 1303.721,A -85,B 0,C 180,E1 2062.1,E2 2062.1} C_VEL
LIN {X 0,Y 576.086,Z 1310.972,A -85,B 0,C 180,E1 2065.496,E2 2065.496} C_VEL
LIN {X 0,Y 576.127,Z 1314.096,A -85,B 0,C 180,E1 2068.502,E2 2068.502} C_VEL
LIN {X 0,Y 576.277,Z 1314.092,A -85,B 0,C 180,E1 2071.503,E2 2071.503} C_VEL
LIN {X 0,Y 576.251,Z 1308.867,A -85,B 0,C 180,E1 2075.702,E2 2075.702} C_VEL
LIN {X 0,Y 576.282,Z 1299.07,A -85,B 0,C 180,E1 2079.422,E2 2079.422} C_VEL
LIN {X 0,Y 576.468,Z 1283.429,A -85,B 0,C 180,E1 2083.244,E2 2083.244} C_VEL
LIN {X 0,Y 576.775,Z 1262.365,A -85,B 0,C 180,E1 2086.921,E2 2086.921} C_VEL
LIN {X 0,Y 577.378,Z 1236.837,A -85,B 0,C 180,E1 2090.265,E2 2090.265} C_VEL
LIN {X 0,Y 578.126,Z 1206.617,A -85,B 0,C 180,E1 2093.304,E2 2093.304} C_VEL
LIN {X 0,Y 579.017,Z 1172.619,A -85,B 0,C 180,E1 2095.903,E2 2095.903} C_VEL
LIN {X 0,Y 579.938,Z 1136.689,A -85,B 0,C 180,E1 2097.932,E2 2097.932} C_VEL
LIN {X 0,Y 580.648,Z 1099.35,A -85,B 0,C 180,E1 2099.402,E2 2099.402} C_VEL
LIN {X 0,Y 581.156,Z 1064.775,A -85,B 0,C 180,E1 2100.249,E2 2100.249} C_VEL
LIN {X 0,Y 580.55,Z 1000.136,A -85,B 0,C 180,E1 2101.221,E2 2101.221} C_VEL
LIN {X 0,Y 575.824,Z 989.03,A -85,B 0,C 180,E1 2101.671,E2 2101.671} C_VEL
LIN {X 0,Y 575.791,Z 989.03,A -85,B 0,C 180,E1 2108.169,E2 2108.169} C_VEL
LIN {X 0,Y 575.811,Z 989.03,A -85,B 0,C 180,E1 2112.957,E2 2112.957} C_VEL
LIN {X 0,Y 575.649,Z 989.03,A -85,B 0,C 180,E1 2119.056,E2 2119.056} C_VEL
LIN {X 0,Y 575.708,Z 989.03,A -85,B 0,C 180,E1 2124.786,E2 2124.786} C_VEL
LIN {X 0,Y 575.821,Z 989.03,A -85,B 0,C 180,E1 2130.139,E2 2130.139} C_VEL
LIN {X 0,Y 575.756,Z 989.03,A -85,B 0,C 180,E1 2135.208,E2 2135.208} C_VEL
LIN {X 0,Y 576.062,Z 989.03,A -85,B 0,C 180,E1 2140.707,E2 2140.707} C_VEL
LIN {X 0,Y 578.083,Z 1003.981,A -85,B 0,C 180,E1 2140.968,E2 2140.968} C_VEL
LIN {X 0,Y 577.874,Z 1036.22,A -85,B 0,C 180,E1 2141.638,E2 2141.638} C_VEL
LIN {X 0,Y 577.528,Z 1066.767,A -85,B 0,C 180,E1 2142.897,E2 2142.897} C_VEL
LIN {X 0,Y 577.178,Z 1093.973,A -85,B 0,C 180,E1 2144.65,E2 2144.65} C_VEL
LIN {X 0,Y 576.719,Z 1118.546,A -85,B 0,C 180,E1 2146.958,E2 2146.958} C_VEL
LIN {X 0,Y 576.467,Z 1138.291,A -85,B 0,C 180,E1 2149.632,E2 2149.632} C_VEL
LIN {X 0,Y 576.326,Z 1152.272,A -85,B 0,C 180,E1 2152.478,E2 2152.478} C_VEL
LIN {X 0,Y 576.272,Z 1161.067,A -85,B 0,C 180,E1 2155.494,E2 2155.494} C_VEL
LIN {X 0,Y 576.264,Z 1164.411,A -85,B 0,C 180,E1 2158.499,E2 2158.499} C_VEL
LIN {X 0,Y 576.311,Z 1162.625,A -85,B 0,C 180,E1 2161.5,E2 2161.5} C_VEL
LIN {X 0,Y 576.346,Z 1155.607,A -85,B 0,C 180,E1 2164.505,E2 2164.505} C_VEL
LIN {X 0,Y 576.477,Z 1142.62,A -85,B 0,C 180,E1 2167.52,E2 2167.52} C_VEL
LIN {X 0,Y 576.727,Z 1123.582,A -85,B 0,C 180,E1 2170.362,E2 2170.362} C_VEL
LIN {X 0,Y 577.031,Z 1100.258,A -85,B 0,C 180,E1 2172.746,E2 2172.746} C_VEL
LIN {X 0,Y 577.469,Z 1072.141,A -85,B 0,C 180,E1 2174.72,E2 2174.72} C_VEL
LIN {X 0,Y 577.865,Z 1042.659,A -85,B 0,C 180,E1 2176.059,E2 2176.059} C_VEL
LIN {X 0,Y 577.926,Z 1010.907,A -85,B 0,C 180,E1 2176.85,E2 2176.85} C_VEL
LIN {X 0,Y 576.078,Z 989.03,A -85,B 0,C 180,E1 2177.234,E2 2177.234} C_VEL
LIN {X 0,Y 575.834,Z 989.03,A -85,B 0,C 180,E1 2183.469,E2 2183.469} C_VEL
LIN {X 0,Y 575.846,Z 989.03,A -85,B 0,C 180,E1 2188.142,E2 2188.142} C_VEL
LIN {X 0,Y 575.89,Z 989.03,A -85,B 0,C 180,E1 2193.383,E2 2193.383} C_VEL
LIN {X 0,Y 575.663,Z 989.03,A -85,B 0,C 180,E1 2198.983,E2 2198.983} C_VEL
LIN {X 0,Y 575.757,Z 989.03,A -85,B 0,C 180,E1 2205.041,E2 2205.041} C_VEL
LIN {X 0,Y 575.759,Z 989.03,A -85,B 0,C 180,E1 2211.017,E2 2211.017} C_VEL
LIN {X 0,Y 575.646,Z 989.03,A -85,B 0,C 180,E1 2216.594,E2 2216.594} C_VEL
LIN {X 0,Y 575.647,Z 989.03,A -85,B 0,C 180,E1 2221.841,E2 2221.841} C_VEL
LIN {X 0,Y 575.625,Z 989.03,A -85,B 0,C 180,E1 2223.074,E2 2223.074} C_VEL
LIN {X 0,Y 579.876,Z 1002.098,A -85,B 0,C 180,E1 2223.485,E2 2223.485} C_VEL
LIN {X 0,Y 579.708,Z 1046.32,A -85,B 0,C 180,E1 2224.263,E2 2224.263} C_VEL
LIN {X 0,Y 579.234,Z 1082.268,A -85,B 0,C 180,E1 2225.492,E2 2225.492} C_VEL
LIN {X 0,Y 578.455,Z 1117.729,A -85,B 0,C 180,E1 2227.343,E2 2227.343} C_VEL
LIN {X 0,Y 577.754,Z 1149.977,A -85,B 0,C 180,E1 2229.726,E2 2229.726} C_VEL
LIN {X 0,Y 577.05,Z 1178.902,A -85,B 0,C 180,E1 2232.608,E2 2232.608} C_VEL
LIN {X 0,Y 576.614,Z 1201.688,A -85,B 0,C 180,E1 2235.653,E2 2235.653} C_VEL
LIN {X 0,Y 576.342,Z 1220.65,A -85,B 0,C 180,E1 2239.122,E2 2239.122} C_VEL
LIN {X 0,Y 576.222,Z 1233.31,A -85,B 0,C 180,E1 2242.473,E2 2242.473} C_VEL
LIN {X 0,Y 576.16,Z 1240.561,A -85,B 0,C 180,E1 2245.49,E2 2245.49} C_VEL
LIN {X 0,Y 576.192,Z 1244.039,A -85,B 0,C 180,E1 2248.496,E2 2248.496} C_VEL
LIN {X 0,Y 576.299,Z 1243.983,A -85,B 0,C 180,E1 2251.498,E2 2251.498} C_VEL
LIN {X 0,Y 576.263,Z 1239.267,A -85,B 0,C 180,E1 2255.078,E2 2255.078} C_VEL
LIN {X 0,Y 576.322,Z 1229.295,A -85,B 0,C 180,E1 2258.656,E2 2258.656} C_VEL
LIN {X 0,Y 576.469,Z 1213.334,A -85,B 0,C 180,E1 2262.277,E2 2262.277} C_VEL
LIN {X 0,Y 576.808,Z 1192.778,A -85,B 0,C 180,E1 2265.552,E2 2265.552} C_VEL
LIN {X 0,Y 577.323,Z 1168.133,A -85,B 0,C 180,E1 2268.475,E2 2268.475} C_VEL
LIN {X 0,Y 578.031,Z 1138.333,A -85,B 0,C 180,E1 2271.134,E2 2271.134} C_VEL
LIN {X 0,Y 578.751,Z 1104.777,A -85,B 0,C 180,E1 2273.322,E2 2273.322} C_VEL
LIN {X 0,Y 579.43,Z 1069.497,A -85,B 0,C 180,E1 2274.924,E2 2274.924} C_VEL
LIN {X 0,Y 579.888,Z 1034.357,A -85,B 0,C 180,E1 2275.921,E2 2275.921} C_VEL
LIN {X 0,Y 579.236,Z 997.956,A -85,B 0,C 180,E1 2276.512,E2 2276.512} C_VEL
LIN {X 0,Y 576.162,Z 989.03,A -85,B 0,C 180,E1 2276.857,E2 2276.857} C_VEL
LIN {X 0,Y 575.872,Z 989.03,A -85,B 0,C 180,E1 2283.384,E2 2283.384} C_VEL
LIN {X 0,Y 575.685,Z 989.03,A -85,B 0,C 180,E1 2288.981,E2 2288.981} C_VEL
LIN {X 0,Y 575.734,Z 989.03,A -85,B 0,C 180,E1 2295.044,E2 2295.044} C_VEL
LIN {X 0,Y 575.748,Z 989.03,A -85,B 0,C 180,E1 2301.024,E2 2301.024} C_VEL
LIN {X 0,Y 575.671,Z 989.03,A -85,B 0,C 180,E1 2306.603,E2 2306.603} C_VEL
LIN {X 0,Y 575.762,Z 989.03,A -85,B 0,C 180,E1 2311.853,E2 2311.853} C_VEL
LIN {X 0,Y 575.721,Z 989.03,A -85,B 0,C 180,E1 2316.85,E2 2316.85} C_VEL
LIN {X 0,Y 575.96,Z 989.03,A -85,B 0,C 180,E1 2321.677,E2 2321.677} C_VEL
LIN {X 0,Y 576.154,Z 989.03,A -85,B 0,C 180,E1 2326.367,E2 2326.367} C_VEL
LIN {X 0,Y 576.01,Z 989.03,A -85,B 0,C 180,E1 2332.671,E2 2332.671} C_VEL
LIN {X 0,Y 576.141,Z 989.03,A -85,B 0,C 180,E1 2336.998,E2 2336.998} C_VEL
LIN {X 0,Y 576.246,Z 989.03,A -85,B 0,C 180,E1 2341.501,E2 2341.501} C_VEL
LIN {X 0,Y 576.23,Z 989.03,A -85,B 0,C 180,E1 2346.013,E2 2346.013} C_VEL
LIN {X 0,Y 575.893,Z 989.03,A -85,B 0,C 180,E1 2349.143,E2 2349.143} C_VEL
LIN {X 0,Y 574.647,Z 989.03,A -85,B 0,C 180,E1 2350.003,E2 2350.003} C_VEL
LIN {X 0,Y 568.046,Z 989.03,A -85,B 0,C 180,E1 2352.344,E2 2352.344} C_VEL
LIN {X 0,Y 567.937,Z 989.03,A -85,B 0,C 180,E1 2352.566,E2 2352.566} C_VEL
LIN {X 0,Y 567.96,Z 989.03,A -85,B 0,C 180,E1 2356.993,E2 2356.993} C_VEL
LIN {X 0,Y 567.902,Z 989.03,A -85,B 0,C 180,E1 2361.838,E2 2361.838} C_VEL
LIN {X 0,Y 567.899,Z 989.03,A -85,B 0,C 180,E1 2366.853,E2 2366.853} C_VEL
LIN {X 0,Y 567.743,Z 989.03,A -85,B 0,C 180,E1 2372.111,E2 2372.111} C_VEL
LIN {X 0,Y 567.905,Z 989.03,A -85,B 0,C 180,E1 2377.671,E2 2377.671} C_VEL
LIN {X 0,Y 567.795,Z 989.03,A -85,B 0,C 180,E1 2383.707,E2 2383.707} C_VEL
LIN {X 0,Y 567.682,Z 989.03,A -85,B 0,C 180,E1 2388.355,E2 2388.355} C_VEL
LIN {X 0,Y 567.739,Z 989.03,A -85,B 0,C 180,E1 2394.217,E2 2394.217} C_VEL
LIN {X 0,Y 568.125,Z 989.123,A -85,B 0,C 180,E1 2397.856,E2 2397.856} C_VEL
LIN {X 0,Y 574.281,Z 1003.749,A -85,B 0,C 180,E1 2398.451,E2 2398.451} C_VEL
LIN {X 0,Y 574.071,Z 1077.541,A -85,B 0,C 180,E1 2399.607,E2 2399.607} C_VEL
LIN {X 0,Y 573.406,Z 1114.758,A -85,B 0,C 180,E1 2400.745,E2 2400.745} C_VEL
LIN {X 0,Y 572.454,Z 1150.848,A -85,B 0,C 180,E1 2402.422,E2 2402.422} C_VEL
LIN {X 0,Y 571.357,Z 1186.138,A -85,B 0,C 180,E1 2404.703,E2 2404.703} C_VEL
LIN {X 0,Y 570.299,Z 1218.568,A -85,B 0,C 180,E1 2407.492,E2 2407.492} C_VEL
LIN {X 0,Y 569.397,Z 1247.656,A -85,B 0,C 180,E1 2410.775,E2 2410.775} C_VEL
LIN {X 0,Y 568.715,Z 1272.078,A -85,B 0,C 180,E1 2414.418,E2 2414.418} C_VEL
LIN {X 0,Y 568.419,Z 1290.454,A -85,B 0,C 180,E1 2418.13,E2 2418.13} C_VEL
LIN {X 0,Y 568.317,Z 1303.721,A -85,B 0,C 180,E1 2421.99,E2 2421.99} C_VEL
LIN {X 0,Y 568.205,Z 1310.974,A -85,B 0,C 180,E1 2425.433,E2 2425.433} C_VEL
LIN {X 0,Y 568.256,Z 1314.099,A -85,B 0,C 180,E1 2428.481,E2 2428.481} C_VEL
LIN {X 0,Y 568.392,Z 1314.094,A -85,B 0,C 180,E1 2431.524,E2 2431.524} C_VEL
LIN {X 0,Y 568.36,Z 1309.357,A -85,B 0,C 180,E1 2435.534,E2 2435.534} C_VEL
LIN {X 0,Y 568.372,Z 1299.073,A -85,B 0,C 180,E1 2439.555,E2 2439.555} C_VEL
LIN {X 0,Y 568.612,Z 1283.424,A -85,B 0,C 180,E1 2443.431,E2 2443.431} C_VEL
LIN {X 0,Y 569.034,Z 1262.111,A -85,B 0,C 180,E1 2447.197,E2 2447.197} C_VEL
LIN {X 0,Y 569.743,Z 1236.837,A -85,B 0,C 180,E1 2450.548,E2 2450.548} C_VEL
LIN {X 0,Y 570.642,Z 1207.116,A -85,B 0,C 180,E1 2453.583,E2 2453.583} C_VEL
LIN {X 0,Y 571.725,Z 1173.653,A -85,B 0,C 180,E1 2456.187,E2 2456.187} C_VEL
LIN {X 0,Y 572.812,Z 1138.32,A -85,B 0,C 180,E1 2458.228,E2 2458.228} C_VEL
LIN {X 0,Y 573.681,Z 1100.684,A -85,B 0,C 180,E1 2459.751,E2 2459.751} C_VEL
LIN {X 0,Y 574.349,Z 1064.796,A -85,B 0,C 180,E1 2460.646,E2 2460.646} C_VEL
LIN {X 0,Y 573.831,Z 1002.705,A -85,B 0,C 180,E1 2461.591,E2 2461.591} C_VEL
LIN {X 0,Y 567.797,Z 989.03,A -85,B 0,C 180,E1 2462.17,E2 2462.17} C_VEL
LIN {X 0,Y 567.902,Z 989.03,A -85,B 0,C 180,E1 2467.678,E2 2467.678} C_VEL
LIN {X 0,Y 567.805,Z 989.03,A -85,B 0,C 180,E1 2473.713,E2 2473.713} C_VEL
LIN {X 0,Y 567.683,Z 989.03,A -85,B 0,C 180,E1 2478.354,E2 2478.354} C_VEL
LIN {X 0,Y 567.736,Z 989.03,A -85,B 0,C 180,E1 2484.216,E2 2484.216} C_VEL
LIN {X 0,Y 567.912,Z 989.03,A -85,B 0,C 180,E1 2489.68,E2 2489.68} C_VEL
LIN {X 0,Y 567.802,Z 989.03,A -85,B 0,C 180,E1 2494.836,E2 2494.836} C_VEL
LIN {X 0,Y 568.124,Z 989.03,A -85,B 0,C 180,E1 2500.445,E2 2500.445} C_VEL
LIN {X 0,Y 570.558,Z 1001.98,A -85,B 0,C 180,E1 2500.696,E2 2500.696} C_VEL
LIN {X 0,Y 570.347,Z 1034.909,A -85,B 0,C 180,E1 2501.361,E2 2501.361} C_VEL
LIN {X 0,Y 569.936,Z 1065.742,A -85,B 0,C 180,E1 2502.624,E2 2502.624} C_VEL
LIN {X 0,Y 569.42,Z 1093.783,A -85,B 0,C 180,E1 2504.436,E2 2504.436} C_VEL
LIN {X 0,Y 568.924,Z 1118.404,A -85,B 0,C 180,E1 2506.776,E2 2506.776} C_VEL
LIN {X 0,Y 568.589,Z 1138.202,A -85,B 0,C 180,E1 2509.487,E2 2509.487} C_VEL
LIN {X 0,Y 568.439,Z 1152.209,A -85,B 0,C 180,E1 2512.373,E2 2512.373} C_VEL
LIN {X 0,Y 568.383,Z 1161.039,A -85,B 0,C 180,E1 2515.432,E2 2515.432} C_VEL
LIN {X 0,Y 568.388,Z 1164.41,A -85,B 0,C 180,E1 2518.478,E2 2518.478} C_VEL
LIN {X 0,Y 568.435,Z 1162.641,A -85,B 0,C 180,E1 2521.521,E2 2521.521} C_VEL
LIN {X 0,Y 568.47,Z 1155.646,A -85,B 0,C 180,E1 2524.567,E2 2524.567} C_VEL
LIN {X 0,Y 568.61,Z 1142.697,A -85,B 0,C 180,E1 2527.625,E2 2527.625} C_VEL
LIN {X 0,Y 568.914,Z 1123.694,A -85,B 0,C 180,E1 2530.506,E2 2530.506} C_VEL
LIN {X 0,Y 569.283,Z 1100.433,A -85,B 0,C 180,E1 2532.923,E2 2532.923} C_VEL
LIN {X 0,Y 569.816,Z 1073.007,A -85,B 0,C 180,E1 2534.886,E2 2534.886} C_VEL
LIN {X 0,Y 570.299,Z 1043.086,A -85,B 0,C 180,E1 2536.278,E2 2536.278} C_VEL
LIN {X 0,Y 570.366,Z 1009.846,A -85,B 0,C 180,E1 2537.112,E2 2537.112} C_VEL
LIN {X 0,Y 568.17,Z 989.03,A -85,B 0,C 180,E1 2537.472,E2 2537.472} C_VEL
LIN {X 0,Y 567.961,Z 989.03,A -85,B 0,C 180,E1 2543.485,E2 2543.485} C_VEL
LIN {X 0,Y 567.841,Z 989.03,A -85,B 0,C 180,E1 2548.713,E2 2548.713} C_VEL
LIN {X 0,Y 567.802,Z 989.03,A -85,B 0,C 180,E1 2554.519,E2 2554.519} C_VEL
LIN {X 0,Y 567.72,Z 989.03,A -85,B 0,C 180,E1 2559.635,E2 2559.635} C_VEL
LIN {X 0,Y 567.793,Z 989.03,A -85,B 0,C 180,E1 2565.851,E2 2565.851} C_VEL
LIN {X 0,Y 567.828,Z 989.03,A -85,B 0,C 180,E1 2570.411,E2 2570.411} C_VEL
LIN {X 0,Y 567.719,Z 989.03,A -85,B 0,C 180,E1 2575.481,E2 2575.481} C_VEL
LIN {X 0,Y 567.829,Z 989.03,A -85,B 0,C 180,E1 2579.669,E2 2579.669} C_VEL
LIN {X 0,Y 567.703,Z 989.033,A -85,B 0,C 180,E1 2582.69,E2 2582.69} C_VEL
LIN {X 0,Y 572.791,Z 1003.156,A -85,B 0,C 180,E1 2583.146,E2 2583.146} C_VEL
LIN {X 0,Y 572.571,Z 1046.182,A -85,B 0,C 180,E1 2583.915,E2 2583.915} C_VEL
LIN {X 0,Y 571.964,Z 1081.661,A -85,B 0,C 180,E1 2585.134,E2 2585.134} C_VEL
LIN {X 0,Y 571.089,Z 1116.534,A -85,B 0,C 180,E1 2586.961,E2 2586.961} C_VEL
LIN {X 0,Y 570.221,Z 1149.095,A -85,B 0,C 180,E1 2589.368,E2 2589.368} C_VEL
LIN {X 0,Y 569.437,Z 1177.137,A -85,B 0,C 180,E1 2592.165,E2 2592.165} C_VEL
LIN {X 0,Y 568.807,Z 1201.686,A -85,B 0,C 180,E1 2595.452,E2 2595.452} C_VEL
LIN {X 0,Y 568.481,Z 1220.516,A -85,B 0,C 180,E1 2598.94,E2 2598.94} C_VEL
LIN {X 0,Y 568.332,Z 1233.308,A -85,B 0,C 180,E1 2602.368,E2 2602.368} C_VEL
LIN {X 0,Y 568.283,Z 1240.56,A -85,B 0,C 180,E1 2605.428,E2 2605.428} C_VEL
LIN {X 0,Y 568.316,Z 1244.039,A -85,B 0,C 180,E1 2608.476,E2 2608.476} C_VEL
LIN {X 0,Y 568.415,Z 1243.983,A -85,B 0,C 180,E1 2611.518,E2 2611.518} C_VEL
LIN {X 0,Y 568.422,Z 1240.427,A -85,B 0,C 180,E1 2614.565,E2 2614.565} C_VEL
LIN {X 0,Y 568.472,Z 1230.63,A -85,B 0,C 180,E1 2618.392,E2 2618.392} C_VEL
LIN {X 0,Y 568.616,Z 1216.225,A -85,B 0,C 180,E1 2621.876,E2 2621.876} C_VEL
LIN {X 0,Y 568.987,Z 1196.901,A -85,B 0,C 180,E1 2625.177,E2 2625.177} C_VEL
LIN {X 0,Y 569.617,Z 1171.52,A -85,B 0,C 180,E1 2628.376,E2 2628.376} C_VEL
LIN {X 0,Y 570.443,Z 1142.078,A -85,B 0,C 180,E1 2631.124,E2 2631.124} C_VEL
LIN {X 0,Y 571.306,Z 1110.061,A -85,B 0,C 180,E1 2633.338,E2 2633.338} C_VEL
LIN {X 0,Y 572.129,Z 1073.866,A -85,B 0,C 180,E1 2635.097,E2 2635.097} C_VEL
LIN {X 0,Y 572.74,Z 1036.762,A -85,B 0,C 180,E1 2636.218,E2 2636.218} C_VEL
LIN {X 0,Y 572.356,Z 1000.476,A -85,B 0,C 180,E1 2636.822,E2 2636.822} C_VEL
LIN {X 0,Y 568.179,Z 989.03,A -85,B 0,C 180,E1 2637.231,E2 2637.231} C_VEL
LIN {X 0,Y 567.858,Z 989.03,A -85,B 0,C 180,E1 2643.918,E2 2643.918} C_VEL
LIN {X 0,Y 567.741,Z 989.03,A -85,B 0,C 180,E1 2649.633,E2 2649.633} C_VEL
LIN {X 0,Y 567.774,Z 989.03,A -85,B 0,C 180,E1 2655.854,E2 2655.854} C_VEL
LIN {X 0,Y 567.839,Z 989.03,A -85,B 0,C 180,E1 2660.411,E2 2660.411} C_VEL
LIN {X 0,Y 567.727,Z 989.03,A -85,B 0,C 180,E1 2665.482,E2 2665.482} C_VEL
LIN {X 0,Y 567.808,Z 989.03,A -85,B 0,C 180,E1 2671.281,E2 2671.281} C_VEL
LIN {X 0,Y 567.839,Z 989.03,A -85,B 0,C 180,E1 2676.51,E2 2676.51} C_VEL
LIN {X 0,Y 568.081,Z 989.03,A -85,B 0,C 180,E1 2681.413,E2 2681.413} C_VEL
LIN {X 0,Y 568.232,Z 989.03,A -85,B 0,C 180,E1 2686.173,E2 2686.173} C_VEL
LIN {X 0,Y 568.082,Z 989.03,A -85,B 0,C 180,E1 2692.657,E2 2692.657} C_VEL
LIN {X 0,Y 568.235,Z 989.03,A -85,B 0,C 180,E1 2696.956,E2 2696.956} C_VEL
LIN {X 0,Y 568.359,Z 989.03,A -85,B 0,C 180,E1 2701.522,E2 2701.522} C_VEL
LIN {X 0,Y 568.296,Z 989.03,A -85,B 0,C 180,E1 2706.097,E2 2706.097} C_VEL
LIN {X 0,Y 567.97,Z 989.03,A -85,B 0,C 180,E1 2712.271,E2 2712.271} C_VEL
LIN {X 0,Y 567.937,Z 989.03,A -85,B 0,C 180,E1 2712.566,E2 2712.566} C_VEL
LIN {X 0,Y 563.999,Z 989.03,A -85,B 0,C 180,E1 2714.288,E2 2714.288} C_VEL
LIN {X 0,Y 560.029,Z 989.03,A -85,B 0,C 180,E1 2716.033,E2 2716.033} C_VEL
LIN {X 0,Y 560.049,Z 989.03,A -85,B 0,C 180,E1 2720.503,E2 2720.503} C_VEL
LIN {X 0,Y 560.01,Z 989.03,A -85,B 0,C 180,E1 2725.539,E2 2725.539} C_VEL
LIN {X 0,Y 559.887,Z 989.03,A -85,B 0,C 180,E1 2730.802,E2 2730.802} C_VEL
LIN {X 0,Y 559.951,Z 989.03,A -85,B 0,C 180,E1 2736.36,E2 2736.36} C_VEL
LIN {X 0,Y 559.893,Z 989.03,A -85,B 0,C 180,E1 2742.359,E2 2742.359} C_VEL
LIN {X 0,Y 559.759,Z 989.03,A -85,B 0,C 180,E1 2747.629,E2 2747.629} C_VEL
LIN {X 0,Y 559.838,Z 989.03,A -85,B 0,C 180,E1 2753.959,E2 2753.959} C_VEL
LIN {X 0,Y 560.221,Z 989.128,A -85,B 0,C 180,E1 2757.346,E2 2757.346} C_VEL
LIN {X 0,Y 567.594,Z 1008.18,A -85,B 0,C 180,E1 2758.101,E2 2758.101} C_VEL
LIN {X 0,Y 567.223,Z 1079.292,A -85,B 0,C 180,E1 2759.243,E2 2759.243} C_VEL
LIN {X 0,Y 566.358,Z 1118.373,A -85,B 0,C 180,E1 2760.489,E2 2760.489} C_VEL
LIN {X 0,Y 565.178,Z 1156.332,A -85,B 0,C 180,E1 2762.355,E2 2762.355} C_VEL
LIN {X 0,Y 563.795,Z 1191.866,A -85,B 0,C 180,E1 2764.788,E2 2764.788} C_VEL
LIN {X 0,Y 562.602,Z 1224.04,A -85,B 0,C 180,E1 2767.738,E2 2767.738} C_VEL
LIN {X 0,Y 561.594,Z 1251.71,A -85,B 0,C 180,E1 2771.048,E2 2771.048} C_VEL
LIN {X 0,Y 560.903,Z 1274.961,A -85,B 0,C 180,E1 2774.724,E2 2774.724} C_VEL
LIN {X 0,Y 560.536,Z 1292.01,A -85,B 0,C 180,E1 2778.354,E2 2778.354} C_VEL
LIN {X 0,Y 560.455,Z 1303.72,A -85,B 0,C 180,E1 2781.877,E2 2781.877} C_VEL
LIN {X 0,Y 560.315,Z 1310.977,A -85,B 0,C 180,E1 2785.369,E2 2785.369} C_VEL
LIN {X 0,Y 560.355,Z 1314.101,A -85,B 0,C 180,E1 2788.46,E2 2788.46} C_VEL
LIN {X 0,Y 560.486,Z 1314.096,A -85,B 0,C 180,E1 2791.546,E2 2791.546} C_VEL
LIN {X 0,Y 560.481,Z 1309.817,A -85,B 0,C 180,E1 2795.366,E2 2795.366} C_VEL
LIN {X 0,Y 560.515,Z 1300.282,A -85,B 0,C 180,E1 2799.299,E2 2799.299} C_VEL
LIN {X 0,Y 560.785,Z 1285.283,A -85,B 0,C 180,E1 2803.226,E2 2803.226} C_VEL
LIN {X 0,Y 561.241,Z 1263.648,A -85,B 0,C 180,E1 2807.207,E2 2807.207} C_VEL
LIN {X 0,Y 562.078,Z 1238.56,A -85,B 0,C 180,E1 2810.636,E2 2810.636} C_VEL
LIN {X 0,Y 563.19,Z 1207.965,A -85,B 0,C 180,E1 2813.837,E2 2813.837} C_VEL
LIN {X 0,Y 564.491,Z 1173.658,A -85,B 0,C 180,E1 2816.549,E2 2816.549} C_VEL
LIN {X 0,Y 565.77,Z 1138.421,A -85,B 0,C 180,E1 2818.607,E2 2818.607} C_VEL
LIN {X 0,Y 566.757,Z 1101.043,A -85,B 0,C 180,E1 2820.14,E2 2820.14} C_VEL
LIN {X 0,Y 567.576,Z 1063.348,A -85,B 0,C 180,E1 2821.077,E2 2821.077} C_VEL
LIN {X 0,Y 566.916,Z 1005.159,A -85,B 0,C 180,E1 2821.986,E2 2821.986} C_VEL
LIN {X 0,Y 559.826,Z 989.03,A -85,B 0,C 180,E1 2822.718,E2 2822.718} C_VEL
LIN {X 0,Y 559.911,Z 989.03,A -85,B 0,C 180,E1 2828.312,E2 2828.312} C_VEL
LIN {X 0,Y 559.865,Z 989.03,A -85,B 0,C 180,E1 2833.306,E2 2833.306} C_VEL
LIN {X 0,Y 559.756,Z 989.03,A -85,B 0,C 180,E1 2839.017,E2 2839.017} C_VEL
LIN {X 0,Y 559.94,Z 989.03,A -85,B 0,C 180,E1 2845.534,E2 2845.534} C_VEL
LIN {X 0,Y 559.963,Z 989.03,A -85,B 0,C 180,E1 2850.984,E2 2850.984} C_VEL
LIN {X 0,Y 560.012,Z 989.03,A -85,B 0,C 180,E1 2856.383,E2 2856.383} C_VEL
LIN {X 0,Y 560.157,Z 989.03,A -85,B 0,C 180,E1 2860.17,E2 2860.17} C_VEL
LIN {X 0,Y 563.071,Z 1002.806,A -85,B 0,C 180,E1 2860.455,E2 2860.455} C_VEL
LIN {X 0,Y 562.808,Z 1035.232,A -85,B 0,C 180,E1 2861.128,E2 2861.128} C_VEL
LIN {X 0,Y 562.296,Z 1066.655,A -85,B 0,C 180,E1 2862.444,E2 2862.444} C_VEL
LIN {X 0,Y 561.682,Z 1094.832,A -85,B 0,C 180,E1 2864.316,E2 2864.316} C_VEL
LIN {X 0,Y 561.151,Z 1118.263,A -85,B 0,C 180,E1 2866.589,E2 2866.589} C_VEL
LIN {X 0,Y 560.736,Z 1138.113,A -85,B 0,C 180,E1 2869.338,E2 2869.338} C_VEL
LIN {X 0,Y 560.554,Z 1152.145,A -85,B 0,C 180,E1 2872.265,E2 2872.265} C_VEL
LIN {X 0,Y 560.479,Z 1161.011,A -85,B 0,C 180,E1 2875.367,E2 2875.367} C_VEL
LIN {X 0,Y 560.486,Z 1164.408,A -85,B 0,C 180,E1 2878.457,E2 2878.457} C_VEL
LIN {X 0,Y 560.535,Z 1162.657,A -85,B 0,C 180,E1 2881.542,E2 2881.542} C_VEL
LIN {X 0,Y 560.581,Z 1155.685,A -85,B 0,C 180,E1 2884.632,E2 2884.632} C_VEL
LIN {X 0,Y 560.769,Z 1142.774,A -85,B 0,C 180,E1 2887.732,E2 2887.732} C_VEL
LIN {X 0,Y 561.112,Z 1123.8,A -85,B 0,C 180,E1 2890.654,E2 2890.654} C_VEL
LIN {X 0,Y 561.544,Z 1100.607,A -85,B 0,C 180,E1 2893.104,E2 2893.104} C_VEL
LIN {X 0,Y 562.193,Z 1073.035,A -85,B 0,C 180,E1 2895.107,E2 2895.107} C_VEL
LIN {X 0,Y 562.74,Z 1043.514,A -85,B 0,C 180,E1 2896.502,E2 2896.502} C_VEL
LIN {X 0,Y 562.883,Z 1010.807,A -85,B 0,C 180,E1 2897.346,E2 2897.346} C_VEL
LIN {X 0,Y 560.891,Z 992.074,A -85,B 0,C 180,E1 2897.671,E2 2897.671} C_VEL
LIN {X 0,Y 560.273,Z 989.03,A -85,B 0,C 180,E1 2897.802,E2 2897.802} C_VEL
LIN {X 0,Y 560.004,Z 989.03,A -85,B 0,C 180,E1 2903.839,E2 2903.839} C_VEL
LIN {X 0,Y 559.9,Z 989.03,A -85,B 0,C 180,E1 2909.019,E2 2909.019} C_VEL
LIN {X 0,Y 559.922,Z 989.03,A -85,B 0,C 180,E1 2914.467,E2 2914.467} C_VEL
LIN {X 0,Y 559.75,Z 989.03,A -85,B 0,C 180,E1 2920.982,E2 2920.982} C_VEL
LIN {X 0,Y 559.859,Z 989.03,A -85,B 0,C 180,E1 2926.694,E2 2926.694} C_VEL
LIN {X 0,Y 559.919,Z 989.03,A -85,B 0,C 180,E1 2931.689,E2 2931.689} C_VEL
LIN {X 0,Y 559.799,Z 989.03,A -85,B 0,C 180,E1 2937.371,E2 2937.371} C_VEL
LIN {X 0,Y 559.789,Z 989.03,A -85,B 0,C 180,E1 2942.23,E2 2942.23} C_VEL
LIN {X 0,Y 565.824,Z 1007.314,A -85,B 0,C 180,E1 2942.848,E2 2942.848} C_VEL
LIN {X 0,Y 565.447,Z 1047.816,A -85,B 0,C 180,E1 2943.607,E2 2943.607} C_VEL
LIN {X 0,Y 564.714,Z 1084.241,A -85,B 0,C 180,E1 2944.909,E2 2944.909} C_VEL
LIN {X 0,Y 563.585,Z 1119.903,A -85,B 0,C 180,E1 2946.859,E2 2946.859} C_VEL
LIN {X 0,Y 562.59,Z 1151.365,A -85,B 0,C 180,E1 2949.281,E2 2949.281} C_VEL
LIN {X 0,Y 561.635,Z 1179.649,A -85,B 0,C 180,E1 2952.204,E2 2952.204} C_VEL
LIN {X 0,Y 560.989,Z 1203.468,A -85,B 0,C 180,E1 2955.539,E2 2955.539} C_VEL
LIN {X 0,Y 560.617,Z 1220.339,A -85,B 0,C 180,E1 2958.743,E2 2958.743} C_VEL
LIN {X 0,Y 560.451,Z 1233.307,A -85,B 0,C 180,E1 2962.26,E2 2962.26} C_VEL
LIN {X 0,Y 560.391,Z 1240.559,A -85,B 0,C 180,E1 2965.363,E2 2965.363} C_VEL
LIN {X 0,Y 560.414,Z 1244.039,A -85,B 0,C 180,E1 2968.454,E2 2968.454} C_VEL
LIN {X 0,Y 560.511,Z 1243.984,A -85,B 0,C 180,E1 2971.54,E2 2971.54} C_VEL
LIN {X 0,Y 560.438,Z 1238.92,A -85,B 0,C 180,E1 2975.397,E2 2975.397} C_VEL
LIN {X 0,Y 560.577,Z 1229.301,A -85,B 0,C 180,E1 2978.901,E2 2978.901} C_VEL
LIN {X 0,Y 560.783,Z 1213.346,A -85,B 0,C 180,E1 2982.626,E2 2982.626} C_VEL
LIN {X 0,Y 561.23,Z 1192.782,A -85,B 0,C 180,E1 2985.995,E2 2985.995} C_VEL
LIN {X 0,Y 562.072,Z 1166.948,A -85,B 0,C 180,E1 2989.123,E2 2989.123} C_VEL
LIN {X 0,Y 563.111,Z 1135.695,A -85,B 0,C 180,E1 2991.929,E2 2991.929} C_VEL
LIN {X 0,Y 564.175,Z 1102.531,A -85,B 0,C 180,E1 2994.09,E2 2994.09} C_VEL
LIN {X 0,Y 565.071,Z 1068.474,A -85,B 0,C 180,E1 2995.644,E2 2995.644} C_VEL
LIN {X 0,Y 565.723,Z 1033.56,A -85,B 0,C 180,E1 2996.64,E2 2996.64} C_VEL
LIN {X 0,Y 565.397,Z 1002.87,A -85,B 0,C 180,E1 2997.147,E2 2997.147} C_VEL
LIN {X 0,Y 560.185,Z 989.03,A -85,B 0,C 180,E1 2997.647,E2 2997.647} C_VEL
LIN {X 0,Y 559.91,Z 989.03,A -85,B 0,C 180,E1 3003.339,E2 3003.339} C_VEL
LIN {X 0,Y 559.751,Z 989.03,A -85,B 0,C 180,E1 3008.578,E2 3008.578} C_VEL
LIN {X 0,Y 559.796,Z 989.03,A -85,B 0,C 180,E1 3014.494,E2 3014.494} C_VEL
LIN {X 0,Y 559.863,Z 989.03,A -85,B 0,C 180,E1 3019.696,E2 3019.696} C_VEL
LIN {X 0,Y 559.845,Z 989.03,A -85,B 0,C 180,E1 3025.528,E2 3025.528} C_VEL
LIN {X 0,Y 559.888,Z 989.03,A -85,B 0,C 180,E1 3030.98,E2 3030.98} C_VEL
LIN {X 0,Y 559.931,Z 989.03,A -85,B 0,C 180,E1 3036.387,E2 3036.387} C_VEL
LIN {X 0,Y 560.146,Z 989.03,A -85,B 0,C 180,E1 3041.14,E2 3041.14} C_VEL
LIN {X 0,Y 560.284,Z 989.03,A -85,B 0,C 180,E1 3045.973,E2 3045.973} C_VEL
LIN {X 0,Y 560.178,Z 989.03,A -85,B 0,C 180,E1 3052.645,E2 3052.645} C_VEL
LIN {X 0,Y 560.326,Z 989.03,A -85,B 0,C 180,E1 3056.913,E2 3056.913} C_VEL
LIN {X 0,Y 560.448,Z 989.03,A -85,B 0,C 180,E1 3061.543,E2 3061.543} C_VEL
LIN {X 0,Y 560.376,Z 989.03,A -85,B 0,C 180,E1 3066.184,E2 3066.184} C_VEL
LIN {X 0,Y 560.035,Z 989.03,A -85,B 0,C 180,E1 3072.556,E2 3072.556} C_VEL
LIN {X 0,Y 560.029,Z 989.03,A -85,B 0,C 180,E1 3076.033,E2 3076.033} C_VEL
LIN {X 0,Y 556.038,Z 989.03,A -85,B 0,C 180,E1 3077.777,E2 3077.777} C_VEL
LIN {X 0,Y 552.059,Z 989.03,A -85,B 0,C 180,E1 3079.546,E2 3079.546} C_VEL
LIN {X 0,Y 552.112,Z 989.03,A -85,B 0,C 180,E1 3085.589,E2 3085.589} C_VEL
LIN {X 0,Y 551.899,Z 989.03,A -85,B 0,C 180,E1 3091.297,E2 3091.297} C_VEL
LIN {X 0,Y 551.977,Z 989.03,A -85,B 0,C 180,E1 3097.554,E2 3097.554} C_VEL
LIN {X 0,Y 551.966,Z 989.03,A -85,B 0,C 180,E1 3103.113,E2 3103.113} C_VEL
LIN {X 0,Y 551.875,Z 989.03,A -85,B 0,C 180,E1 3108.989,E2 3108.989} C_VEL
LIN {X 0,Y 551.992,Z 989.03,A -85,B 0,C 180,E1 3115.094,E2 3115.094} C_VEL
LIN {X 0,Y 552.253,Z 989.337,A -85,B 0,C 180,E1 3116.818,E2 3116.818} C_VEL
LIN {X 0,Y 560.877,Z 1010.248,A -85,B 0,C 180,E1 3117.703,E2 3117.703} C_VEL
LIN {X 0,Y 560.41,Z 1079.279,A -85,B 0,C 180,E1 3118.828,E2 3118.828} C_VEL
LIN {X 0,Y 559.441,Z 1118.299,A -85,B 0,C 180,E1 3120.085,E2 3120.085} C_VEL
LIN {X 0,Y 558.027,Z 1156.187,A -85,B 0,C 180,E1 3121.96,E2 3121.96} C_VEL
LIN {X 0,Y 556.425,Z 1193.003,A -85,B 0,C 180,E1 3124.527,E2 3124.527} C_VEL
LIN {X 0,Y 555,Z 1225.515,A -85,B 0,C 180,E1 3127.578,E2 3127.578} C_VEL
LIN {X 0,Y 553.865,Z 1252.75,A -85,B 0,C 180,E1 3130.919,E2 3130.919} C_VEL
LIN {X 0,Y 553.081,Z 1274.78,A -85,B 0,C 180,E1 3134.469,E2 3134.469} C_VEL
LIN {X 0,Y 552.671,Z 1292.013,A -85,B 0,C 180,E1 3138.186,E2 3138.186} C_VEL
LIN {X 0,Y 552.59,Z 1303.719,A -85,B 0,C 180,E1 3141.76,E2 3141.76} C_VEL
LIN {X 0,Y 552.437,Z 1310.979,A -85,B 0,C 180,E1 3145.302,E2 3145.302} C_VEL
LIN {X 0,Y 552.46,Z 1314.103,A -85,B 0,C 180,E1 3148.438,E2 3148.438} C_VEL
LIN {X 0,Y 552.58,Z 1314.098,A -85,B 0,C 180,E1 3151.568,E2 3151.568} C_VEL
LIN {X 0,Y 552.542,Z 1309.359,A -85,B 0,C 180,E1 3155.688,E2 3155.688} C_VEL
LIN {X 0,Y 552.616,Z 1300.28,A -85,B 0,C 180,E1 3159.433,E2 3159.433} C_VEL
LIN {X 0,Y 552.932,Z 1285.286,A -85,B 0,C 180,E1 3163.417,E2 3163.417} C_VEL
LIN {X 0,Y 553.496,Z 1263.644,A -85,B 0,C 180,E1 3167.455,E2 3167.455} C_VEL
LIN {X 0,Y 554.534,Z 1236.827,A -85,B 0,C 180,E1 3171.139,E2 3171.139} C_VEL
LIN {X 0,Y 555.827,Z 1206.502,A -85,B 0,C 180,E1 3174.31,E2 3174.31} C_VEL
LIN {X 0,Y 557.348,Z 1171.993,A -85,B 0,C 180,E1 3177.036,E2 3177.036} C_VEL
LIN {X 0,Y 558.845,Z 1135.095,A -85,B 0,C 180,E1 3179.17,E2 3179.17} C_VEL
LIN {X 0,Y 560.012,Z 1097.329,A -85,B 0,C 180,E1 3180.669,E2 3180.669} C_VEL
LIN {X 0,Y 560.843,Z 1060.16,A -85,B 0,C 180,E1 3181.549,E2 3181.549} C_VEL
LIN {X 0,Y 560.399,Z 1008.044,A -85,B 0,C 180,E1 3182.36,E2 3182.36} C_VEL
LIN {X 0,Y 551.879,Z 989.03,A -85,B 0,C 180,E1 3183.213,E2 3183.213} C_VEL
LIN {X 0,Y 551.969,Z 989.03,A -85,B 0,C 180,E1 3188.966,E2 3188.966} C_VEL
LIN {X 0,Y 551.929,Z 989.03,A -85,B 0,C 180,E1 3194.698,E2 3194.698} C_VEL
LIN {X 0,Y 551.831,Z 989.03,A -85,B 0,C 180,E1 3199.974,E2 3199.974} C_VEL
LIN {X 0,Y 551.995,Z 989.03,A -85,B 0,C 180,E1 3205.105,E2 3205.105} C_VEL
LIN {X 0,Y 552.079,Z 989.03,A -85,B 0,C 180,E1 3211.014,E2 3211.014} C_VEL
LIN {X 0,Y 552.061,Z 989.03,A -85,B 0,C 180,E1 3217.501,E2 3217.501} C_VEL
LIN {X 0,Y 552.205,Z 989.031,A -85,B 0,C 180,E1 3219.892,E2 3219.892} C_VEL
LIN {X 0,Y 555.592,Z 1003.682,A -85,B 0,C 180,E1 3220.209,E2 3220.209} C_VEL
LIN {X 0,Y 555.273,Z 1035.828,A -85,B 0,C 180,E1 3220.897,E2 3220.897} C_VEL
LIN {X 0,Y 554.698,Z 1066.772,A -85,B 0,C 180,E1 3222.218,E2 3222.218} C_VEL
LIN {X 0,Y 554,Z 1094.641,A -85,B 0,C 180,E1 3224.093,E2 3224.093} C_VEL
LIN {X 0,Y 553.324,Z 1119.86,A -85,B 0,C 180,E1 3226.597,E2 3226.597} C_VEL
LIN {X 0,Y 552.864,Z 1138.777,A -85,B 0,C 180,E1 3229.321,E2 3229.321} C_VEL
LIN {X 0,Y 552.676,Z 1152.082,A -85,B 0,C 180,E1 3232.154,E2 3232.154} C_VEL
LIN {X 0,Y 552.597,Z 1160.983,A -85,B 0,C 180,E1 3235.301,E2 3235.301} C_VEL
LIN {X 0,Y 552.588,Z 1164.406,A -85,B 0,C 180,E1 3238.435,E2 3238.435} C_VEL
LIN {X 0,Y 552.637,Z 1162.673,A -85,B 0,C 180,E1 3241.564,E2 3241.564} C_VEL
LIN {X 0,Y 552.706,Z 1155.724,A -85,B 0,C 180,E1 3244.698,E2 3244.698} C_VEL
LIN {X 0,Y 552.901,Z 1142.852,A -85,B 0,C 180,E1 3247.843,E2 3247.843} C_VEL
LIN {X 0,Y 553.274,Z 1124.541,A -85,B 0,C 180,E1 3250.722,E2 3250.722} C_VEL
LIN {X 0,Y 553.788,Z 1101.914,A -85,B 0,C 180,E1 3253.191,E2 3253.191} C_VEL
LIN {X 0,Y 554.514,Z 1074.543,A -85,B 0,C 180,E1 3255.241,E2 3255.241} C_VEL
LIN {X 0,Y 555.184,Z 1045.323,A -85,B 0,C 180,E1 3256.683,E2 3256.683} C_VEL
LIN {X 0,Y 555.458,Z 1014.266,A -85,B 0,C 180,E1 3257.54,E2 3257.54} C_VEL
LIN {X 0,Y 553.74,Z 994.775,A -85,B 0,C 180,E1 3257.886,E2 3257.886} C_VEL
LIN {X 0,Y 552.373,Z 989.03,A -85,B 0,C 180,E1 3258.034,E2 3258.034} C_VEL
LIN {X 0,Y 552.039,Z 989.03,A -85,B 0,C 180,E1 3264.205,E2 3264.205} C_VEL
LIN {X 0,Y 551.966,Z 989.03,A -85,B 0,C 180,E1 3269.477,E2 3269.477} C_VEL
LIN {X 0,Y 551.937,Z 989.03,A -85,B 0,C 180,E1 3275.038,E2 3275.038} C_VEL
LIN {X 0,Y 551.869,Z 989.03,A -85,B 0,C 180,E1 3281.011,E2 3281.011} C_VEL
LIN {X 0,Y 551.97,Z 989.03,A -85,B 0,C 180,E1 3286.879,E2 3286.879} C_VEL
LIN {X 0,Y 551.981,Z 989.03,A -85,B 0,C 180,E1 3293.022,E2 3293.022} C_VEL
LIN {X 0,Y 551.921,Z 989.03,A -85,B 0,C 180,E1 3298.698,E2 3298.698} C_VEL
LIN {X 0,Y 551.925,Z 989.03,A -85,B 0,C 180,E1 3301.836,E2 3301.836} C_VEL
LIN {X 0,Y 558.827,Z 1008.707,A -85,B 0,C 180,E1 3302.499,E2 3302.499} C_VEL
LIN {X 0,Y 558.323,Z 1047.763,A -85,B 0,C 180,E1 3303.243,E2 3303.243} C_VEL
LIN {X 0,Y 557.446,Z 1084.214,A -85,B 0,C 180,E1 3304.559,E2 3304.559} C_VEL
LIN {X 0,Y 556.24,Z 1119.196,A -85,B 0,C 180,E1 3306.486,E2 3306.486} C_VEL
LIN {X 0,Y 555.052,Z 1151.356,A -85,B 0,C 180,E1 3308.986,E2 3308.986} C_VEL
LIN {X 0,Y 553.948,Z 1180.261,A -85,B 0,C 180,E1 3312.025,E2 3312.025} C_VEL
LIN {X 0,Y 553.192,Z 1203.467,A -85,B 0,C 180,E1 3315.33,E2 3315.33} C_VEL
LIN {X 0,Y 552.768,Z 1220.338,A -85,B 0,C 180,E1 3318.581,E2 3318.581} C_VEL
LIN {X 0,Y 552.573,Z 1233.306,A -85,B 0,C 180,E1 3322.149,E2 3322.149} C_VEL
LIN {X 0,Y 552.517,Z 1240.558,A -85,B 0,C 180,E1 3325.297,E2 3325.297} C_VEL
LIN {X 0,Y 552.516,Z 1244.039,A -85,B 0,C 180,E1 3328.432,E2 3328.432} C_VEL
LIN {X 0,Y 552.606,Z 1243.985,A -85,B 0,C 180,E1 3331.562,E2 3331.562} C_VEL
LIN {X 0,Y 552.563,Z 1239.639,A -85,B 0,C 180,E1 3335.109,E2 3335.109} C_VEL
LIN {X 0,Y 552.714,Z 1230.633,A -85,B 0,C 180,E1 3338.633,E2 3338.633} C_VEL
LIN {X 0,Y 552.891,Z 1216.281,A -85,B 0,C 180,E1 3342.209,E2 3342.209} C_VEL
LIN {X 0,Y 553.409,Z 1197.419,A -85,B 0,C 180,E1 3345.539,E2 3345.539} C_VEL
LIN {X 0,Y 554.261,Z 1171.93,A -85,B 0,C 180,E1 3348.86,E2 3348.86} C_VEL
LIN {X 0,Y 555.431,Z 1142.095,A -85,B 0,C 180,E1 3351.723,E2 3351.723} C_VEL
LIN {X 0,Y 556.621,Z 1110.09,A -85,B 0,C 180,E1 3353.992,E2 3353.992} C_VEL
LIN {X 0,Y 557.731,Z 1074.319,A -85,B 0,C 180,E1 3355.775,E2 3355.775} C_VEL
LIN {X 0,Y 558.594,Z 1037.602,A -85,B 0,C 180,E1 3356.915,E2 3356.915} C_VEL
LIN {X 0,Y 558.092,Z 1004.204,A -85,B 0,C 180,E1 3357.514,E2 3357.514} C_VEL
LIN {X 0,Y 552.205,Z 989.03,A -85,B 0,C 180,E1 3358.123,E2 3358.123} C_VEL
LIN {X 0,Y 552.026,Z 989.03,A -85,B 0,C 180,E1 3363.14,E2 3363.14} C_VEL
LIN {X 0,Y 551.834,Z 989.03,A -85,B 0,C 180,E1 3368.97,E2 3368.97} C_VEL
LIN {X 0,Y 551.896,Z 989.03,A -85,B 0,C 180,E1 3374.695,E2 3374.695} C_VEL
LIN {X 0,Y 551.95,Z 989.03,A -85,B 0,C 180,E1 3379.95,E2 3379.95} C_VEL
LIN {X 0,Y 551.95,Z 989.03,A -85,B 0,C 180,E1 3385.101,E2 3385.101} C_VEL
LIN {X 0,Y 551.983,Z 989.03,A -85,B 0,C 180,E1 3391.02,E2 3391.02} C_VEL
LIN {X 0,Y 552.015,Z 989.03,A -85,B 0,C 180,E1 3395.794,E2 3395.794} C_VEL
LIN {X 0,Y 552.232,Z 989.03,A -85,B 0,C 180,E1 3400.859,E2 3400.859} C_VEL
LIN {X 0,Y 552.368,Z 989.03,A -85,B 0,C 180,E1 3405.768,E2 3405.768} C_VEL
LIN {X 0,Y 552.335,Z 989.03,A -85,B 0,C 180,E1 3412.149,E2 3412.149} C_VEL
LIN {X 0,Y 552.427,Z 989.03,A -85,B 0,C 180,E1 3416.869,E2 3416.869} C_VEL
LIN {X 0,Y 552.539,Z 989.03,A -85,B 0,C 180,E1 3421.565,E2 3421.565} C_VEL
LIN {X 0,Y 552.445,Z 989.03,A -85,B 0,C 180,E1 3426.273,E2 3426.273} C_VEL
LIN {X 0,Y 552.135,Z 989.03,A -85,B 0,C 180,E1 3432.629,E2 3432.629} C_VEL
LIN {X 0,Y 552.109,Z 989.03,A -85,B 0,C 180,E1 3437.496,E2 3437.496} C_VEL
LIN {X 0,Y 552.059,Z 989.03,A -85,B 0,C 180,E1 3439.546,E2 3439.546} C_VEL
LIN {X 0,Y 548.052,Z 989.03,A -85,B 0,C 180,E1 3441.316,E2 3441.316} C_VEL
LIN {X 0,Y 544.061,Z 989.03,A -85,B 0,C 180,E1 3443.112,E2 3443.112} C_VEL
LIN {X 0,Y 544.073,Z 989.03,A -85,B 0,C 180,E1 3448.131,E2 3448.131} C_VEL
LIN {X 0,Y 543.938,Z 989.03,A -85,B 0,C 180,E1 3453.699,E2 3453.699} C_VEL
LIN {X 0,Y 544.039,Z 989.03,A -85,B 0,C 180,E1 3459.638,E2 3459.638} C_VEL
LIN {X 0,Y 544.002,Z 989.03,A -85,B 0,C 180,E1 3463.904,E2 3463.904} C_VEL
LIN {X 0,Y 543.922,Z 989.03,A -85,B 0,C 180,E1 3470.353,E2 3470.353} C_VEL
LIN {X 0,Y 544.289,Z 989.685,A -85,B 0,C 180,E1 3476.274,E2 3476.274} C_VEL
LIN {X 0,Y 554.202,Z 1011.955,A -85,B 0,C 180,E1 3477.292,E2 3477.292} C_VEL
LIN {X 0,Y 553.644,Z 1079.121,A -85,B 0,C 180,E1 3478.4,E2 3478.4} C_VEL
LIN {X 0,Y 552.496,Z 1118.434,A -85,B 0,C 180,E1 3479.676,E2 3479.676} C_VEL
LIN {X 0,Y 550.951,Z 1155.93,A -85,B 0,C 180,E1 3481.552,E2 3481.552} C_VEL
LIN {X 0,Y 549.167,Z 1192.352,A -85,B 0,C 180,E1 3484.11,E2 3484.11} C_VEL
LIN {X 0,Y 547.555,Z 1224.041,A -85,B 0,C 180,E1 3487.093,E2 3487.093} C_VEL
LIN {X 0,Y 546.248,Z 1251.376,A -85,B 0,C 180,E1 3490.445,E2 3490.445} C_VEL
LIN {X 0,Y 545.293,Z 1274.26,A -85,B 0,C 180,E1 3494.143,E2 3494.143} C_VEL
LIN {X 0,Y 544.83,Z 1292.017,A -85,B 0,C 180,E1 3498.014,E2 3498.014} C_VEL
LIN {X 0,Y 544.712,Z 1303.718,A -85,B 0,C 180,E1 3501.64,E2 3501.64} C_VEL
LIN {X 0,Y 544.538,Z 1310.982,A -85,B 0,C 180,E1 3505.234,E2 3505.234} C_VEL
LIN {X 0,Y 544.559,Z 1314.105,A -85,B 0,C 180,E1 3508.415,E2 3508.415} C_VEL
LIN {X 0,Y 544.673,Z 1314.1,A -85,B 0,C 180,E1 3511.591,E2 3511.591} C_VEL
LIN {X 0,Y 544.654,Z 1309.726,A -85,B 0,C 180,E1 3515.568,E2 3515.568} C_VEL
LIN {X 0,Y 544.718,Z 1300.277,A -85,B 0,C 180,E1 3519.571,E2 3519.571} C_VEL
LIN {X 0,Y 545.099,Z 1285.447,A -85,B 0,C 180,E1 3523.577,E2 3523.577} C_VEL
LIN {X 0,Y 545.788,Z 1263.641,A -85,B 0,C 180,E1 3527.71,E2 3527.71} C_VEL
LIN {X 0,Y 546.938,Z 1237.07,A -85,B 0,C 180,E1 3531.416,E2 3531.416} C_VEL
LIN {X 0,Y 548.4,Z 1207.04,A -85,B 0,C 180,E1 3534.61,E2 3534.61} C_VEL
LIN {X 0,Y 550.07,Z 1173.664,A -85,B 0,C 180,E1 3537.302,E2 3537.302} C_VEL
LIN {X 0,Y 551.783,Z 1136.714,A -85,B 0,C 180,E1 3539.494,E2 3539.494} C_VEL
LIN {X 0,Y 553.102,Z 1099.683,A -85,B 0,C 180,E1 3541.012,E2 3541.012} C_VEL
LIN {X 0,Y 554.107,Z 1061.688,A -85,B 0,C 180,E1 3541.95,E2 3541.95} C_VEL
LIN {X 0,Y 553.562,Z 1010.373,A -85,B 0,C 180,E1 3542.775,E2 3542.775} C_VEL
LIN {X 0,Y 543.952,Z 989.03,A -85,B 0,C 180,E1 3543.802,E2 3543.802} C_VEL
LIN {X 0,Y 544.035,Z 989.03,A -85,B 0,C 180,E1 3549.645,E2 3549.645} C_VEL
LIN {X 0,Y 544.028,Z 989.03,A -85,B 0,C 180,E1 3553.909,E2 3553.909} C_VEL
LIN {X 0,Y 543.909,Z 989.03,A -85,B 0,C 180,E1 3560.351,E2 3560.351} C_VEL
LIN {X 0,Y 544.11,Z 989.03,A -85,B 0,C 180,E1 3566.313,E2 3566.313} C_VEL
LIN {X 0,Y 544.085,Z 989.03,A -85,B 0,C 180,E1 3571.87,E2 3571.87} C_VEL
LIN {X 0,Y 544.111,Z 989.03,A -85,B 0,C 180,E1 3577.154,E2 3577.154} C_VEL
LIN {X 0,Y 544.282,Z 989.03,A -85,B 0,C 180,E1 3579.58,E2 3579.58} C_VEL
LIN {X 0,Y 548.113,Z 1005.923,A -85,B 0,C 180,E1 3579.974,E2 3579.974} C_VEL
LIN {X 0,Y 547.741,Z 1037.395,A -85,B 0,C 180,E1 3580.696,E2 3580.696} C_VEL
LIN {X 0,Y 547.05,Z 1068.241,A -85,B 0,C 180,E1 3582.058,E2 3582.058} C_VEL
LIN {X 0,Y 546.278,Z 1095.623,A -85,B 0,C 180,E1 3583.965,E2 3583.965} C_VEL
LIN {X 0,Y 545.552,Z 1119.719,A -85,B 0,C 180,E1 3586.402,E2 3586.402} C_VEL
LIN {X 0,Y 545.013,Z 1138.689,A -85,B 0,C 180,E1 3589.165,E2 3589.165} C_VEL
LIN {X 0,Y 544.803,Z 1152.019,A -85,B 0,C 180,E1 3592.04,E2 3592.04} C_VEL
LIN {X 0,Y 544.717,Z 1160.955,A -85,B 0,C 180,E1 3595.233,E2 3595.233} C_VEL
LIN {X 0,Y 544.686,Z 1164.404,A -85,B 0,C 180,E1 3598.412,E2 3598.412} C_VEL
LIN {X 0,Y 544.738,Z 1162.689,A -85,B 0,C 180,E1 3601.587,E2 3601.587} C_VEL
LIN {X 0,Y 544.824,Z 1155.763,A -85,B 0,C 180,E1 3604.766,E2 3604.766} C_VEL
LIN {X 0,Y 545.039,Z 1142.929,A -85,B 0,C 180,E1 3607.956,E2 3607.956} C_VEL
LIN {X 0,Y 545.448,Z 1124.648,A -85,B 0,C 180,E1 3610.877,E2 3610.877} C_VEL
LIN {X 0,Y 546.052,Z 1102.088,A -85,B 0,C 180,E1 3613.381,E2 3613.381} C_VEL
LIN {X 0,Y 546.881,Z 1075.006,A -85,B 0,C 180,E1 3615.444,E2 3615.444} C_VEL
LIN {X 0,Y 547.645,Z 1045.532,A -85,B 0,C 180,E1 3616.927,E2 3616.927} C_VEL
LIN {X 0,Y 547.993,Z 1015.107,A -85,B 0,C 180,E1 3617.787,E2 3617.787} C_VEL
LIN {X 0,Y 546.236,Z 996.151,A -85,B 0,C 180,E1 3618.137,E2 3618.137} C_VEL
LIN {X 0,Y 544.456,Z 989.03,A -85,B 0,C 180,E1 3618.363,E2 3618.363} C_VEL
LIN {X 0,Y 544.11,Z 989.03,A -85,B 0,C 180,E1 3624.581,E2 3624.581} C_VEL
LIN {X 0,Y 543.991,Z 989.03,A -85,B 0,C 180,E1 3630.683,E2 3630.683} C_VEL
LIN {X 0,Y 543.926,Z 989.03,A -85,B 0,C 180,E1 3635.631,E2 3635.631} C_VEL
LIN {X 0,Y 543.943,Z 989.03,A -85,B 0,C 180,E1 3641.742,E2 3641.742} C_VEL
LIN {X 0,Y 544.049,Z 989.03,A -85,B 0,C 180,E1 3648.26,E2 3648.26} C_VEL
LIN {X 0,Y 544.005,Z 989.03,A -85,B 0,C 180,E1 3654.367,E2 3654.367} C_VEL
LIN {X 0,Y 544.032,Z 989.03,A -85,B 0,C 180,E1 3660.566,E2 3660.566} C_VEL
LIN {X 0,Y 543.999,Z 989.154,A -85,B 0,C 180,E1 3661.397,E2 3661.397} C_VEL
LIN {X 0,Y 551.814,Z 1009.922,A -85,B 0,C 180,E1 3662.138,E2 3662.138} C_VEL
LIN {X 0,Y 551.247,Z 1049.002,A -85,B 0,C 180,E1 3662.909,E2 3662.909} C_VEL
LIN {X 0,Y 550.231,Z 1085.63,A -85,B 0,C 180,E1 3664.268,E2 3664.268} C_VEL
LIN {X 0,Y 548.797,Z 1121.107,A -85,B 0,C 180,E1 3666.284,E2 3666.284} C_VEL
LIN {X 0,Y 547.481,Z 1152.477,A -85,B 0,C 180,E1 3668.788,E2 3668.788} C_VEL
LIN {X 0,Y 546.22,Z 1181.236,A -85,B 0,C 180,E1 3671.889,E2 3671.889} C_VEL
LIN {X 0,Y 545.364,Z 1204.962,A -85,B 0,C 180,E1 3675.372,E2 3675.372} C_VEL
LIN {X 0,Y 544.876,Z 1222.061,A -85,B 0,C 180,E1 3678.818,E2 3678.818} C_VEL
LIN {X 0,Y 544.68,Z 1234.44,A -85,B 0,C 180,E1 3682.435,E2 3682.435} C_VEL
LIN {X 0,Y 544.668,Z 1241.433,A -85,B 0,C 180,E1 3685.814,E2 3685.814} C_VEL
LIN {X 0,Y 544.564,Z 1244.497,A -85,B 0,C 180,E1 3689.997,E2 3689.997} C_VEL
LIN {X 0,Y 544.67,Z 1242.633,A -85,B 0,C 180,E1 3693.173,E2 3693.173} C_VEL
LIN {X 0,Y 544.736,Z 1235.305,A -85,B 0,C 180,E1 3697.158,E2 3697.158} C_VEL
LIN {X 0,Y 544.982,Z 1221.707,A -85,B 0,C 180,E1 3701.173,E2 3701.173} C_VEL
LIN {X 0,Y 545.512,Z 1203.521,A -85,B 0,C 180,E1 3704.781,E2 3704.781} C_VEL
LIN {X 0,Y 546.34,Z 1180.593,A -85,B 0,C 180,E1 3708.101,E2 3708.101} C_VEL
LIN {X 0,Y 547.471,Z 1152.715,A -85,B 0,C 180,E1 3711.1,E2 3711.1} C_VEL
LIN {X 0,Y 548.797,Z 1121.444,A -85,B 0,C 180,E1 3713.602,E2 3713.602} C_VEL
LIN {X 0,Y 550.119,Z 1087.053,A -85,B 0,C 180,E1 3715.581,E2 3715.581} C_VEL
LIN {X 0,Y 551.198,Z 1049.184,A -85,B 0,C 180,E1 3716.998,E2 3716.998} C_VEL
LIN {X 0,Y 551.567,Z 1007.58,A -85,B 0,C 180,E1 3717.819,E2 3717.819} C_VEL
LIN {X 0,Y 544.243,Z 989.03,A -85,B 0,C 180,E1 3718.558,E2 3718.558} C_VEL
LIN {X 0,Y 544.072,Z 989.03,A -85,B 0,C 180,E1 3723.693,E2 3723.693} C_VEL
LIN {X 0,Y 543.911,Z 989.03,A -85,B 0,C 180,E1 3729.648,E2 3729.648} C_VEL
LIN {X 0,Y 544,Z 989.03,A -85,B 0,C 180,E1 3736.152,E2 3736.152} C_VEL
LIN {X 0,Y 544.086,Z 989.03,A -85,B 0,C 180,E1 3742.401,E2 3742.401} C_VEL
LIN {X 0,Y 544.029,Z 989.03,A -85,B 0,C 180,E1 3748.198,E2 3748.198} C_VEL
LIN {X 0,Y 544.099,Z 989.03,A -85,B 0,C 180,E1 3753.659,E2 3753.659} C_VEL
LIN {X 0,Y 544.222,Z 989.03,A -85,B 0,C 180,E1 3758.873,E2 3758.873} C_VEL
LIN {X 0,Y 544.298,Z 989.03,A -85,B 0,C 180,E1 3763.906,E2 3763.906} C_VEL
LIN {X 0,Y 544.264,Z 989.03,A -85,B 0,C 180,E1 3768.81,E2 3768.81} C_VEL
LIN {X 0,Y 544.33,Z 989.03,A -85,B 0,C 180,E1 3773.634,E2 3773.634} C_VEL
LIN {X 0,Y 544.302,Z 989.03,A -85,B 0,C 180,E1 3778.412,E2 3778.412} C_VEL
LIN {X 0,Y 544.34,Z 989.03,A -85,B 0,C 180,E1 3783.178,E2 3783.178} C_VEL
LIN {X 0,Y 544.255,Z 989.03,A -85,B 0,C 180,E1 3787.969,E2 3787.969} C_VEL
LIN {X 0,Y 544.216,Z 989.03,A -85,B 0,C 180,E1 3792.816,E2 3792.816} C_VEL
LIN {X 0,Y 544.178,Z 989.03,A -85,B 0,C 180,E1 3797.759,E2 3797.759} C_VEL
LIN {X 0,Y 544.061,Z 989.03,A -85,B 0,C 180,E1 3803.112,E2 3803.112} C_VEL
LIN {X 0,Y 542.774,Z 989.03,A -85,B 0,C 180,E1 3804.024,E2 3804.024} C_VEL
LIN {X 0,Y 536.239,Z 989.03,A -85,B 0,C 180,E1 3806.51,E2 3806.51} C_VEL
LIN {X 0,Y 536.17,Z 989.03,A -85,B 0,C 180,E1 3806.745,E2 3806.745} C_VEL
LIN {X 0,Y 536.011,Z 989.03,A -85,B 0,C 180,E1 3812.377,E2 3812.377} C_VEL
LIN {X 0,Y 536.145,Z 989.03,A -85,B 0,C 180,E1 3818.256,E2 3818.256} C_VEL
LIN {X 0,Y 535.98,Z 989.03,A -85,B 0,C 180,E1 3824.735,E2 3824.735} C_VEL
LIN {X 0,Y 535.962,Z 989.03,A -85,B 0,C 180,E1 3829.644,E2 3829.644} C_VEL
LIN {X 0,Y 536.046,Z 989.111,A -85,B 0,C 180,E1 3834.015,E2 3834.015} C_VEL
LIN {X 0,Y 537.766,Z 993.873,A -85,B 0,C 180,E1 3834.816,E2 3834.816} C_VEL
LIN {X 0,Y 539.444,Z 996.637,A -85,B 0,C 180,E1 3835.984,E2 3835.984} C_VEL
LIN {X 0,Y 547.422,Z 1013.534,A -85,B 0,C 180,E1 3836.859,E2 3836.859} C_VEL
LIN {X 0,Y 546.908,Z 1079.107,A -85,B 0,C 180,E1 3837.965,E2 3837.965} C_VEL
LIN {X 0,Y 545.656,Z 1117.924,A -85,B 0,C 180,E1 3839.232,E2 3839.232} C_VEL
LIN {X 0,Y 543.914,Z 1155.161,A -85,B 0,C 180,E1 3841.101,E2 3841.101} C_VEL
LIN {X 0,Y 541.912,Z 1191.427,A -85,B 0,C 180,E1 3843.656,E2 3843.656} C_VEL
LIN {X 0,Y 540.088,Z 1224.035,A -85,B 0,C 180,E1 3846.758,E2 3846.758} C_VEL
LIN {X 0,Y 538.584,Z 1251.38,A -85,B 0,C 180,E1 3850.155,E2 3850.155} C_VEL
LIN {X 0,Y 537.494,Z 1274.259,A -85,B 0,C 180,E1 3853.907,E2 3853.907} C_VEL
LIN {X 0,Y 536.978,Z 1292.02,A -85,B 0,C 180,E1 3857.836,E2 3857.836} C_VEL
LIN {X 0,Y 536.813,Z 1303.717,A -85,B 0,C 180,E1 3861.516,E2 3861.516} C_VEL
LIN {X 0,Y 536.641,Z 1310.985,A -85,B 0,C 180,E1 3865.164,E2 3865.164} C_VEL
LIN {X 0,Y 536.668,Z 1314.107,A -85,B 0,C 180,E1 3868.392,E2 3868.392} C_VEL
LIN {X 0,Y 536.797,Z 1314.102,A -85,B 0,C 180,E1 3871.614,E2 3871.614} C_VEL
LIN {X 0,Y 536.757,Z 1309.722,A -85,B 0,C 180,E1 3875.65,E2 3875.65} C_VEL
LIN {X 0,Y 536.828,Z 1300.274,A -85,B 0,C 180,E1 3879.713,E2 3879.713} C_VEL
LIN {X 0,Y 537.254,Z 1285.761,A -85,B 0,C 180,E1 3883.705,E2 3883.705} C_VEL
LIN {X 0,Y 537.95,Z 1265.635,A -85,B 0,C 180,E1 3887.632,E2 3887.632} C_VEL
LIN {X 0,Y 539.205,Z 1240.273,A -85,B 0,C 180,E1 3891.339,E2 3891.339} C_VEL
LIN {X 0,Y 540.953,Z 1208.351,A -85,B 0,C 180,E1 3894.846,E2 3894.846} C_VEL
LIN {X 0,Y 542.847,Z 1174.696,A -85,B 0,C 180,E1 3897.62,E2 3897.62} C_VEL
LIN {X 0,Y 544.75,Z 1138.318,A -85,B 0,C 180,E1 3899.826,E2 3899.826} C_VEL
LIN {X 0,Y 546.243,Z 1101.718,A -85,B 0,C 180,E1 3901.374,E2 3901.374} C_VEL
LIN {X 0,Y 547.376,Z 1063.623,A -85,B 0,C 180,E1 3902.356,E2 3902.356} C_VEL
LIN {X 0,Y 546.994,Z 1013.16,A -85,B 0,C 180,E1 3903.176,E2 3903.176} C_VEL
LIN {X 0,Y 539.334,Z 996.937,A -85,B 0,C 180,E1 3904.032,E2 3904.032} C_VEL
LIN {X 0,Y 536.532,Z 991.69,A -85,B 0,C 180,E1 3905.67,E2 3905.67} C_VEL
LIN {X 0,Y 536.092,Z 989.03,A -85,B 0,C 180,E1 3906.113,E2 3906.113} C_VEL
LIN {X 0,Y 536.08,Z 989.03,A -85,B 0,C 180,E1 3910.537,E2 3910.537} C_VEL
LIN {X 0,Y 535.993,Z 989.03,A -85,B 0,C 180,E1 3915.267,E2 3915.267} C_VEL
LIN {X 0,Y 535.974,Z 989.03,A -85,B 0,C 180,E1 3921.729,E2 3921.729} C_VEL
LIN {X 0,Y 536.186,Z 989.03,A -85,B 0,C 180,E1 3927.676,E2 3927.676} C_VEL
LIN {X 0,Y 536.114,Z 989.03,A -85,B 0,C 180,E1 3933.235,E2 3933.235} C_VEL
LIN {X 0,Y 536.37,Z 989.03,A -85,B 0,C 180,E1 3939.292,E2 3939.292} C_VEL
LIN {X 0,Y 540.657,Z 1006.02,A -85,B 0,C 180,E1 3939.703,E2 3939.703} C_VEL
LIN {X 0,Y 540.207,Z 1038.404,A -85,B 0,C 180,E1 3940.469,E2 3940.469} C_VEL
LIN {X 0,Y 539.437,Z 1069.243,A -85,B 0,C 180,E1 3941.868,E2 3941.868} C_VEL
LIN {X 0,Y 538.543,Z 1096.604,A -85,B 0,C 180,E1 3943.833,E2 3943.833} C_VEL
LIN {X 0,Y 537.79,Z 1119.577,A -85,B 0,C 180,E1 3946.202,E2 3946.202} C_VEL
LIN {X 0,Y 537.196,Z 1138.143,A -85,B 0,C 180,E1 3948.92,E2 3948.92} C_VEL
LIN {X 0,Y 536.932,Z 1151.955,A -85,B 0,C 180,E1 3951.922,E2 3951.922} C_VEL
LIN {X 0,Y 536.815,Z 1160.927,A -85,B 0,C 180,E1 3955.162,E2 3955.162} C_VEL
LIN {X 0,Y 536.793,Z 1164.402,A -85,B 0,C 180,E1 3958.389,E2 3958.389} C_VEL
LIN {X 0,Y 536.87,Z 1162.705,A -85,B 0,C 180,E1 3961.61,E2 3961.61} C_VEL
LIN {X 0,Y 536.936,Z 1155.802,A -85,B 0,C 180,E1 3964.836,E2 3964.836} C_VEL
LIN {X 0,Y 537.177,Z 1143.006,A -85,B 0,C 180,E1 3968.074,E2 3968.074} C_VEL
LIN {X 0,Y 537.651,Z 1124.105,A -85,B 0,C 180,E1 3971.127,E2 3971.127} C_VEL
LIN {X 0,Y 538.384,Z 1101.129,A -85,B 0,C 180,E1 3973.679,E2 3973.679} C_VEL
LIN {X 0,Y 539.333,Z 1072.788,A -85,B 0,C 180,E1 3975.825,E2 3975.825} C_VEL
LIN {X 0,Y 540.15,Z 1043.144,A -85,B 0,C 180,E1 3977.275,E2 3977.275} C_VEL
